LIN {X 0,Y 258.894,Z 466.884,A -85,B 0,C 180,E1 -21997.54,E2 -21997.54} C_VEL
LIN {X 0,Y 258.497,Z 472.697,A -85,B 0,C 180,E1 -21997.806,E2 -21997.806} C_VEL
LIN {X 0,Y 256.025,Z 487.683,A -85,B 0,C 180,E1 -21997.807,E2 -21997.807} C_VEL
LIN {X 0,Y 255.441,Z 492.024,A -85,B 0,C 180,E1 -21997.871,E2 -21997.871} C_VEL
LIN {X 0,Y 249.944,Z 542.974,A -85,B 0,C 180,E1 -21999.352,E2 -21999.352} C_VEL
LIN {X 0,Y 247.16,Z 558.513,A -85,B 0,C 180,E1 -22000.006,E2 -22000.006} C_VEL
LIN {X 0,Y 243.376,Z 573.661,A -85,B 0,C 180,E1 -22000.867,E2 -22000.867} C_VEL
LIN {X 0,Y 238.802,Z 588.296,A -85,B 0,C 180,E1 -22002.002,E2 -22002.002} C_VEL
LIN {X 0,Y 233.418,Z 602.419,A -85,B 0,C 180,E1 -22003.415,E2 -22003.415} C_VEL
LIN {X 0,Y 227.735,Z 615.394,A -85,B 0,C 180,E1 -22005.11,E2 -22005.11} C_VEL
LIN {X 0,Y 221.851,Z 627.382,A -85,B 0,C 180,E1 -22007.08,E2 -22007.08} C_VEL
LIN {X 0,Y 215.808,Z 638.427,A -85,B 0,C 180,E1 -22009.358,E2 -22009.358} C_VEL
LIN {X 0,Y 209.362,Z 649.302,A -85,B 0,C 180,E1 -22012.219,E2 -22012.219} C_VEL
LIN {X 0,Y 202.723,Z 659.642,A -85,B 0,C 180,E1 -22015.711,E2 -22015.711} C_VEL
LIN {X 0,Y 197.738,Z 667.198,A -85,B 0,C 180,E1 -22018.978,E2 -22018.978} C_VEL
LIN {X 0,Y 192.862,Z 674.32,A -85,B 0,C 180,E1 -22022.901,E2 -22022.901} C_VEL
LIN {X 0,Y 188.983,Z 680.037,A -85,B 0,C 180,E1 -22027.015,E2 -22027.015} C_VEL
LIN {X 0,Y 186.775,Z 683.529,A -85,B 0,C 180,E1 -22030.204,E2 -22030.204} C_VEL
LIN {X 0,Y 184.668,Z 687.065,A -85,B 0,C 180,E1 -22034.549,E2 -22034.549} C_VEL
LIN {X 0,Y 183.499,Z 689.425,A -85,B 0,C 180,E1 -22038.959,E2 -22038.959} C_VEL
LIN {X 0,Y 183.209,Z 690.67,A -85,B 0,C 180,E1 -22043.391,E2 -22043.391} C_VEL
LIN {X 0,Y 183.489,Z 690.777,A -85,B 0,C 180,E1 -22047.804,E2 -22047.804} C_VEL
LIN {X 0,Y 183.575,Z 690.376,A -85,B 0,C 180,E1 -22049.999,E2 -22049.999} C_VEL
LIN {X 0,Y 183.501,Z 689.635,A -85,B 0,C 180,E1 -22052.194,E2 -22052.194} C_VEL
LIN {X 0,Y 183.393,Z 688.283,A -85,B 0,C 180,E1 -22054.89,E2 -22054.89} C_VEL
LIN {X 0,Y 183.468,Z 684.438,A -85,B 0,C 180,E1 -22059.925,E2 -22059.925} C_VEL
LIN {X 0,Y 184.277,Z 679.597,A -85,B 0,C 180,E1 -22064.352,E2 -22064.352} C_VEL
LIN {X 0,Y 185.905,Z 673.547,A -85,B 0,C 180,E1 -22068.553,E2 -22068.553} C_VEL
LIN {X 0,Y 188.14,Z 666.3,A -85,B 0,C 180,E1 -22072.512,E2 -22072.512} C_VEL
LIN {X 0,Y 191.186,Z 657.896,A -85,B 0,C 180,E1 -22076.174,E2 -22076.174} C_VEL
LIN {X 0,Y 194.447,Z 648.32,A -85,B 0,C 180,E1 -22079.564,E2 -22079.564} C_VEL
LIN {X 0,Y 198.437,Z 637.302,A -85,B 0,C 180,E1 -22082.69,E2 -22082.69} C_VEL
LIN {X 0,Y 202.681,Z 624.904,A -85,B 0,C 180,E1 -22085.506,E2 -22085.506} C_VEL
LIN {X 0,Y 207.036,Z 611.105,A -85,B 0,C 180,E1 -22087.97,E2 -22087.97} C_VEL
LIN {X 0,Y 210.313,Z 599.494,A -85,B 0,C 180,E1 -22089.627,E2 -22089.627} C_VEL
LIN {X 0,Y 213.614,Z 586.184,A -85,B 0,C 180,E1 -22091.147,E2 -22091.147} C_VEL
LIN {X 0,Y 216.705,Z 571.321,A -85,B 0,C 180,E1 -22092.451,E2 -22092.451} C_VEL
LIN {X 0,Y 219.017,Z 556.883,A -85,B 0,C 180,E1 -22093.384,E2 -22093.384} C_VEL
LIN {X 0,Y 220.649,Z 541.441,A -85,B 0,C 180,E1 -22094.086,E2 -22094.086} C_VEL
LIN {X 0,Y 226.58,Z 457.676,A -85,B 0,C 180,E1 -22096.818,E2 -22096.818} C_VEL
LIN {X 0,Y 221.97,Z 445.741,A -85,B 0,C 180,E1 -22098.326,E2 -22098.326} C_VEL
LIN {X 0,Y 214.721,Z 429.117,A -85,B 0,C 180,E1 -22100.794,E2 -22100.794} C_VEL
LIN {X 0,Y 207.931,Z 415.232,A -85,B 0,C 180,E1 -22103.211,E2 -22103.211} C_VEL
LIN {X 0,Y 200.809,Z 401.844,A -85,B 0,C 180,E1 -22105.947,E2 -22105.947} C_VEL
LIN {X 0,Y 194.594,Z 391.34,A -85,B 0,C 180,E1 -22108.497,E2 -22108.497} C_VEL
LIN {X 0,Y 191.128,Z 385.801,A -85,B 0,C 180,E1 -22110.01,E2 -22110.01} C_VEL
LIN {X 0,Y 189.077,Z 382.495,A -85,B 0,C 180,E1 -22110.953,E2 -22110.953} C_VEL
LIN {X 0,Y 186.429,Z 379.541,A -85,B 0,C 180,E1 -22112.116,E2 -22112.116} C_VEL
LIN {X 0,Y 185.553,Z 376.999,A -85,B 0,C 180,E1 -22112.662,E2 -22112.662} C_VEL
LIN {X 0,Y 185.585,Z 376.991,A -85,B 0,C 180,E1 -22115.383,E2 -22115.383} C_VEL
LIN {X 0,Y 185.672,Z 376.976,A -85,B 0,C 180,E1 -22121.133,E2 -22121.133} C_VEL
LIN {X 0,Y 185.717,Z 376.979,A -85,B 0,C 180,E1 -22124.64,E2 -22124.64} C_VEL
LIN {X 0,Y 185.921,Z 376.902,A -85,B 0,C 180,E1 -22129.36,E2 -22129.36} C_VEL
LIN {X 0,Y 185.958,Z 376.943,A -85,B 0,C 180,E1 -22133.491,E2 -22133.491} C_VEL
LIN {X 0,Y 186.206,Z 376.889,A -85,B 0,C 180,E1 -22137.838,E2 -22137.838} C_VEL
LIN {X 0,Y 186.405,Z 376.87,A -85,B 0,C 180,E1 -22140.001,E2 -22140.001} C_VEL
LIN {X 0,Y 185.925,Z 376.943,A -85,B 0,C 180,E1 -22144.337,E2 -22144.337} C_VEL
LIN {X 0,Y 186.022,Z 376.915,A -85,B 0,C 180,E1 -22148.693,E2 -22148.693} C_VEL
LIN {X 0,Y 185.763,Z 376.965,A -85,B 0,C 180,E1 -22153.121,E2 -22153.121} C_VEL
LIN {X 0,Y 185.673,Z 376.968,A -85,B 0,C 180,E1 -22158.867,E2 -22158.867} C_VEL
LIN {X 0,Y 185.576,Z 376.965,A -85,B 0,C 180,E1 -22164.647,E2 -22164.647} C_VEL
LIN {X 0,Y 185.578,Z 376.992,A -85,B 0,C 180,E1 -22169.494,E2 -22169.494} C_VEL
LIN {X 0,Y 185.499,Z 376.973,A -85,B 0,C 180,E1 -22174.633,E2 -22174.633} C_VEL
LIN {X 0,Y 185.505,Z 376.99,A -85,B 0,C 180,E1 -22177.314,E2 -22177.314} C_VEL
LIN {X 0,Y 185.47,Z 377.001,A -85,B 0,C 180,E1 -22180.726,E2 -22180.726} C_VEL
LIN {X 0,Y 185.459,Z 377.003,A -85,B 0,C 180,E1 -22186.057,E2 -22186.057} C_VEL
LIN {X 0,Y 185.467,Z 376.991,A -85,B 0,C 180,E1 -22189.896,E2 -22189.896} C_VEL
LIN {X 0,Y 185.506,Z 376.986,A -85,B 0,C 180,E1 -22192.713,E2 -22192.713} C_VEL
LIN {X 0,Y 185.534,Z 376.98,A -85,B 0,C 180,E1 -22197.974,E2 -22197.974} C_VEL
LIN {X 0,Y 185.552,Z 376.994,A -85,B 0,C 180,E1 -22200.595,E2 -22200.595} C_VEL
LIN {X 0,Y 185.582,Z 376.98,A -85,B 0,C 180,E1 -22205.383,E2 -22205.383} C_VEL
LIN {X 0,Y 185.594,Z 377.186,A -85,B 0,C 180,E1 -22208.538,E2 -22208.538} C_VEL
LIN {X 0,Y 186.504,Z 379.774,A -85,B 0,C 180,E1 -22209.065,E2 -22209.065} C_VEL
LIN {X 0,Y 188.589,Z 381.975,A -85,B 0,C 180,E1 -22209.979,E2 -22209.979} C_VEL
LIN {X 0,Y 189.237,Z 382.799,A -85,B 0,C 180,E1 -22210.265,E2 -22210.265} C_VEL
LIN {X 0,Y 191.446,Z 386.042,A -85,B 0,C 180,E1 -22211.243,E2 -22211.243} C_VEL
LIN {X 0,Y 192.728,Z 387.647,A -85,B 0,C 180,E1 -22211.774,E2 -22211.774} C_VEL
LIN {X 0,Y 196.707,Z 393.467,A -85,B 0,C 180,E1 -22213.436,E2 -22213.436} C_VEL
LIN {X 0,Y 202.066,Z 401.068,A -85,B 0,C 180,E1 -22215.492,E2 -22215.492} C_VEL
LIN {X 0,Y 208.644,Z 411.142,A -85,B 0,C 180,E1 -22217.858,E2 -22217.858} C_VEL
LIN {X 0,Y 218.699,Z 428.297,A -85,B 0,C 180,E1 -22221.182,E2 -22221.182} C_VEL
LIN {X 0,Y 224.077,Z 439.264,A -85,B 0,C 180,E1 -22222.896,E2 -22222.896} C_VEL
LIN {X 0,Y 226.692,Z 444.585,A -85,B 0,C 180,E1 -22223.685,E2 -22223.685} C_VEL
LIN {X 0,Y 221.003,Z 525.158,A -85,B 0,C 180,E1 -22226.354,E2 -22226.354} C_VEL
LIN {X 0,Y 219.241,Z 540.282,A -85,B 0,C 180,E1 -22227.158,E2 -22227.158} C_VEL
LIN {X 0,Y 216.778,Z 556.065,A -85,B 0,C 180,E1 -22228.375,E2 -22228.375} C_VEL
LIN {X 0,Y 213.955,Z 569.884,A -85,B 0,C 180,E1 -22229.766,E2 -22229.766} C_VEL
LIN {X 0,Y 210.61,Z 583.889,A -85,B 0,C 180,E1 -22231.582,E2 -22231.582} C_VEL
LIN {X 0,Y 207.012,Z 596.7,A -85,B 0,C 180,E1 -22233.651,E2 -22233.651} C_VEL
LIN {X 0,Y 203,Z 609.426,A -85,B 0,C 180,E1 -22236.212,E2 -22236.212} C_VEL
LIN {X 0,Y 199.238,Z 620.577,A -85,B 0,C 180,E1 -22238.995,E2 -22238.995} C_VEL
LIN {X 0,Y 195.131,Z 631.811,A -85,B 0,C 180,E1 -22242.481,E2 -22242.481} C_VEL
LIN {X 0,Y 191.905,Z 640.574,A -85,B 0,C 180,E1 -22245.855,E2 -22245.855} C_VEL
LIN {X 0,Y 189.074,Z 648.331,A -85,B 0,C 180,E1 -22249.545,E2 -22249.545} C_VEL
LIN {X 0,Y 186.876,Z 654.596,A -85,B 0,C 180,E1 -22253.26,E2 -22253.26} C_VEL
LIN {X 0,Y 185.27,Z 659.746,A -85,B 0,C 180,E1 -22257.079,E2 -22257.079} C_VEL
LIN {X 0,Y 184.026,Z 663.921,A -85,B 0,C 180,E1 -22261.037,E2 -22261.037} C_VEL
LIN {X 0,Y 183.21,Z 667.1,A -85,B 0,C 180,E1 -22265.129,E2 -22265.129} C_VEL
LIN {X 0,Y 183.007,Z 669.413,A -85,B 0,C 180,E1 -22269.819,E2 -22269.819} C_VEL
LIN {X 0,Y 183.291,Z 670.312,A -85,B 0,C 180,E1 -22273.646,E2 -22273.646} C_VEL
LIN {X 0,Y 183.797,Z 670.444,A -85,B 0,C 180,E1 -22276.597,E2 -22276.597} C_VEL
LIN {X 0,Y 184.616,Z 670.065,A -85,B 0,C 180,E1 -22279.671,E2 -22279.671} C_VEL
LIN {X 0,Y 185.823,Z 669.085,A -85,B 0,C 180,E1 -22282.76,E2 -22282.76} C_VEL
LIN {X 0,Y 188.251,Z 666.631,A -85,B 0,C 180,E1 -22287.225,E2 -22287.225} C_VEL
LIN {X 0,Y 191.654,Z 662.78,A -85,B 0,C 180,E1 -22291.654,E2 -22291.654} C_VEL
LIN {X 0,Y 195.826,Z 657.743,A -85,B 0,C 180,E1 -22295.762,E2 -22295.762} C_VEL
LIN {X 0,Y 200.527,Z 651.657,A -85,B 0,C 180,E1 -22299.483,E2 -22299.483} C_VEL
LIN {X 0,Y 205.875,Z 644.351,A -85,B 0,C 180,E1 -22302.912,E2 -22302.912} C_VEL
LIN {X 0,Y 211.587,Z 635.885,A -85,B 0,C 180,E1 -22306.055,E2 -22306.055} C_VEL
LIN {X 0,Y 217.343,Z 626.565,A -85,B 0,C 180,E1 -22308.812,E2 -22308.812} C_VEL
LIN {X 0,Y 223.561,Z 615.487,A -85,B 0,C 180,E1 -22311.394,E2 -22311.394} C_VEL
LIN {X 0,Y 229.638,Z 603.29,A -85,B 0,C 180,E1 -22313.63,E2 -22313.63} C_VEL
LIN {X 0,Y 235.175,Z 590.54,A -85,B 0,C 180,E1 -22315.5,E2 -22315.5} C_VEL
LIN {X 0,Y 239.706,Z 578.249,A -85,B 0,C 180,E1 -22316.957,E2 -22316.957} C_VEL
LIN {X 0,Y 244.067,Z 564.231,A -85,B 0,C 180,E1 -22318.246,E2 -22318.246} C_VEL
LIN {X 0,Y 247.639,Z 549.484,A -85,B 0,C 180,E1 -22319.311,E2 -22319.311} C_VEL
LIN {X 0,Y 250.324,Z 534.829,A -85,B 0,C 180,E1 -22320.074,E2 -22320.074} C_VEL
LIN {X 0,Y 252.627,Z 516.015,A -85,B 0,C 180,E1 -22320.717,E2 -22320.717} C_VEL
LIN {X 0,Y 258.11,Z 463.213,A -85,B 0,C 180,E1 -22322.272,E2 -22322.272} C_VEL
LIN {X 0,Y 255.837,Z 458.618,A -85,B 0,C 180,E1 -22323.825,E2 -22323.825} C_VEL
LIN {X 0,Y 252.805,Z 452.119,A -85,B 0,C 180,E1 -22326.308,E2 -22326.308} C_VEL
LIN {X 0,Y 251.193,Z 449.368,A -85,B 0,C 180,E1 -22327.778,E2 -22327.778} C_VEL
LIN {X 0,Y 249.475,Z 446.388,A -85,B 0,C 180,E1 -22329.598,E2 -22329.598} C_VEL
LIN {X 0,Y 247.451,Z 442.793,A -85,B 0,C 180,E1 -22332.401,E2 -22332.401} C_VEL
LIN {X 0,Y 245.547,Z 439.936,A -85,B 0,C 180,E1 -22336.85,E2 -22336.85} C_VEL
LIN {X 0,Y 245.453,Z 439.014,A -85,B 0,C 180,E1 -22337.934,E2 -22337.934} C_VEL
LIN {X 0,Y 245.363,Z 440.064,A -85,B 0,C 180,E1 -22341.586,E2 -22341.586} C_VEL
LIN {X 0,Y 245.757,Z 441.035,A -85,B 0,C 180,E1 -22343.381,E2 -22343.381} C_VEL
LIN {X 0,Y 247.729,Z 446.1,A -85,B 0,C 180,E1 -22347.687,E2 -22347.687} C_VEL
LIN {X 0,Y 250.076,Z 451.667,A -85,B 0,C 180,E1 -22350.753,E2 -22350.753} C_VEL
LIN {X 0,Y 252.319,Z 457.376,A -85,B 0,C 180,E1 -22353.055,E2 -22353.055} C_VEL
LIN {X 0,Y 254.622,Z 463.714,A -85,B 0,C 180,E1 -22355.098,E2 -22355.098} C_VEL
LIN {X 0,Y 257.449,Z 472.109,A -85,B 0,C 180,E1 -22357.257,E2 -22357.257} C_VEL
LIN {X 0,Y 257.008,Z 477.164,A -85,B 0,C 180,E1 -22357.446,E2 -22357.446} C_VEL
LIN {X 0,Y 255.441,Z 492.024,A -85,B 0,C 180,E1 -22357.871,E2 -22357.871} C_VEL
LIN {X 0,Y 254.506,Z 497.876,A -85,B 0,C 180,E1 -22357.886,E2 -22357.886} C_VEL
LIN {X 0,Y 249.984,Z 516.998,A -85,B 0,C 180,E1 -22357.218,E2 -22357.218} C_VEL
LIN {X 0,Y 249.146,Z 522.826,A -85,B 0,C 180,E1 -22357.28,E2 -22357.28} C_VEL
LIN {X 0,Y 246.488,Z 544.542,A -85,B 0,C 180,E1 -22357.949,E2 -22357.949} C_VEL
LIN {X 0,Y 243.261,Z 560.781,A -85,B 0,C 180,E1 -22358.651,E2 -22358.651} C_VEL
LIN {X 0,Y 239.213,Z 575.71,A -85,B 0,C 180,E1 -22359.536,E2 -22359.536} C_VEL
LIN {X 0,Y 234.206,Z 590.658,A -85,B 0,C 180,E1 -22360.737,E2 -22360.737} C_VEL
LIN {X 0,Y 228.684,Z 604.269,A -85,B 0,C 180,E1 -22362.147,E2 -22362.147} C_VEL
LIN {X 0,Y 222.387,Z 617.794,A -85,B 0,C 180,E1 -22363.99,E2 -22363.99} C_VEL
LIN {X 0,Y 215.697,Z 630.347,A -85,B 0,C 180,E1 -22366.18,E2 -22366.18} C_VEL
LIN {X 0,Y 208.568,Z 642.468,A -85,B 0,C 180,E1 -22368.921,E2 -22368.921} C_VEL
LIN {X 0,Y 202.013,Z 652.619,A -85,B 0,C 180,E1 -22371.864,E2 -22371.864} C_VEL
LIN {X 0,Y 196.098,Z 661.158,A -85,B 0,C 180,E1 -22375.009,E2 -22375.009} C_VEL
LIN {X 0,Y 190.324,Z 669.289,A -85,B 0,C 180,E1 -22378.87,E2 -22378.87} C_VEL
LIN {X 0,Y 185.374,Z 675.928,A -85,B 0,C 180,E1 -22382.937,E2 -22382.937} C_VEL
LIN {X 0,Y 181.546,Z 681.214,A -85,B 0,C 180,E1 -22387.224,E2 -22387.224} C_VEL
LIN {X 0,Y 178.786,Z 685.274,A -85,B 0,C 180,E1 -22391.67,E2 -22391.67} C_VEL
LIN {X 0,Y 176.947,Z 688.139,A -85,B 0,C 180,E1 -22396.212,E2 -22396.212} C_VEL
LIN {X 0,Y 176.208,Z 689.84,A -85,B 0,C 180,E1 -22400.819,E2 -22400.819} C_VEL
LIN {X 0,Y 176.26,Z 690.43,A -85,B 0,C 180,E1 -22405.425,E2 -22405.425} C_VEL
LIN {X 0,Y 176.394,Z 690.291,A -85,B 0,C 180,E1 -22407.716,E2 -22407.716} C_VEL
LIN {X 0,Y 176.51,Z 689.846,A -85,B 0,C 180,E1 -22409.999,E2 -22409.999} C_VEL
LIN {X 0,Y 176.411,Z 689.074,A -85,B 0,C 180,E1 -22412.282,E2 -22412.282} C_VEL
LIN {X 0,Y 176.324,Z 687.819,A -85,B 0,C 180,E1 -22414.829,E2 -22414.829} C_VEL
LIN {X 0,Y 176.326,Z 684.745,A -85,B 0,C 180,E1 -22419.173,E2 -22419.173} C_VEL
LIN {X 0,Y 177.002,Z 680.138,A -85,B 0,C 180,E1 -22423.781,E2 -22423.781} C_VEL
LIN {X 0,Y 178.651,Z 674.057,A -85,B 0,C 180,E1 -22428.342,E2 -22428.342} C_VEL
LIN {X 0,Y 181.121,Z 666.318,A -85,B 0,C 180,E1 -22432.831,E2 -22432.831} C_VEL
LIN {X 0,Y 184.232,Z 657.999,A -85,B 0,C 180,E1 -22436.629,E2 -22436.629} C_VEL
LIN {X 0,Y 187.638,Z 648.476,A -85,B 0,C 180,E1 -22440.15,E2 -22440.15} C_VEL
LIN {X 0,Y 191.71,Z 637.625,A -85,B 0,C 180,E1 -22443.358,E2 -22443.358} C_VEL
LIN {X 0,Y 195.682,Z 626.455,A -85,B 0,C 180,E1 -22446.022,E2 -22446.022} C_VEL
LIN {X 0,Y 199.789,Z 614.455,A -85,B 0,C 180,E1 -22448.315,E2 -22448.315} C_VEL
LIN {X 0,Y 203.647,Z 601.464,A -85,B 0,C 180,E1 -22450.32,E2 -22450.32} C_VEL
LIN {X 0,Y 207.234,Z 587.586,A -85,B 0,C 180,E1 -22452.008,E2 -22452.008} C_VEL
LIN {X 0,Y 210.436,Z 572.908,A -85,B 0,C 180,E1 -22453.371,E2 -22453.371} C_VEL
LIN {X 0,Y 213.067,Z 557.48,A -85,B 0,C 180,E1 -22454.418,E2 -22454.418} C_VEL
LIN {X 0,Y 214.774,Z 542.635,A -85,B 0,C 180,E1 -22455.124,E2 -22455.124} C_VEL
LIN {X 0,Y 220.925,Z 459.382,A -85,B 0,C 180,E1 -22457.888,E2 -22457.888} C_VEL
LIN {X 0,Y 212.862,Z 439.507,A -85,B 0,C 180,E1 -22460.691,E2 -22460.691} C_VEL
LIN {X 0,Y 204.972,Z 422.541,A -85,B 0,C 180,E1 -22463.587,E2 -22463.587} C_VEL
LIN {X 0,Y 197.06,Z 407.226,A -85,B 0,C 180,E1 -22466.729,E2 -22466.729} C_VEL
LIN {X 0,Y 190.655,Z 396.248,A -85,B 0,C 180,E1 -22469.479,E2 -22469.479} C_VEL
LIN {X 0,Y 187.522,Z 391.178,A -85,B 0,C 180,E1 -22470.907,E2 -22470.907} C_VEL
LIN {X 0,Y 184.927,Z 387.438,A -85,B 0,C 180,E1 -22472.113,E2 -22472.113} C_VEL
LIN {X 0,Y 182.541,Z 384.257,A -85,B 0,C 180,E1 -22473.258,E2 -22473.258} C_VEL
LIN {X 0,Y 181.864,Z 383.068,A -85,B 0,C 180,E1 -22473.615,E2 -22473.615} C_VEL
LIN {X 0,Y 179.618,Z 380.883,A -85,B 0,C 180,E1 -22474.699,E2 -22474.699} C_VEL
LIN {X 0,Y 178.648,Z 378.396,A -85,B 0,C 180,E1 -22475.289,E2 -22475.289} C_VEL
LIN {X 0,Y 178.542,Z 377.868,A -85,B 0,C 180,E1 -22475.434,E2 -22475.434} C_VEL
LIN {X 0,Y 178.647,Z 377.85,A -85,B 0,C 180,E1 -22481.657,E2 -22481.657} C_VEL
LIN {X 0,Y 178.664,Z 377.83,A -85,B 0,C 180,E1 -22486.349,E2 -22486.349} C_VEL
LIN {X 0,Y 178.935,Z 377.782,A -85,B 0,C 180,E1 -22490.962,E2 -22490.962} C_VEL
LIN {X 0,Y 179.152,Z 377.767,A -85,B 0,C 180,E1 -22497.753,E2 -22497.753} C_VEL
LIN {X 0,Y 179.368,Z 377.745,A -85,B 0,C 180,E1 -22500.001,E2 -22500.001} C_VEL
LIN {X 0,Y 178.873,Z 377.819,A -85,B 0,C 180,E1 -22504.508,E2 -22504.508} C_VEL
LIN {X 0,Y 178.973,Z 377.796,A -85,B 0,C 180,E1 -22509.038,E2 -22509.038} C_VEL
LIN {X 0,Y 178.68,Z 377.842,A -85,B 0,C 180,E1 -22513.651,E2 -22513.651} C_VEL
LIN {X 0,Y 178.621,Z 377.849,A -85,B 0,C 180,E1 -22519.216,E2 -22519.216} C_VEL
LIN {X 0,Y 178.519,Z 377.839,A -85,B 0,C 180,E1 -22525.115,E2 -22525.115} C_VEL
LIN {X 0,Y 178.5,Z 377.875,A -85,B 0,C 180,E1 -22530.788,E2 -22530.788} C_VEL
LIN {X 0,Y 178.484,Z 377.847,A -85,B 0,C 180,E1 -22534.221,E2 -22534.221} C_VEL
LIN {X 0,Y 178.395,Z 377.889,A -85,B 0,C 180,E1 -22539.076,E2 -22539.076} C_VEL
LIN {X 0,Y 178.397,Z 377.866,A -85,B 0,C 180,E1 -22542.047,E2 -22542.047} C_VEL
LIN {X 0,Y 178.393,Z 377.869,A -85,B 0,C 180,E1 -22545.166,E2 -22545.166} C_VEL
LIN {X 0,Y 178.403,Z 377.885,A -85,B 0,C 180,E1 -22548.461,E2 -22548.461} C_VEL
LIN {X 0,Y 178.423,Z 377.881,A -85,B 0,C 180,E1 -22553.784,E2 -22553.784} C_VEL
LIN {X 0,Y 178.485,Z 377.868,A -85,B 0,C 180,E1 -22556.548,E2 -22556.548} C_VEL
LIN {X 0,Y 178.451,Z 377.882,A -85,B 0,C 180,E1 -22561.798,E2 -22561.798} C_VEL
LIN {X 0,Y 178.52,Z 377.862,A -85,B 0,C 180,E1 -22565.737,E2 -22565.737} C_VEL
LIN {X 0,Y 179.413,Z 380.567,A -85,B 0,C 180,E1 -22566.337,E2 -22566.337} C_VEL
LIN {X 0,Y 181.466,Z 382.798,A -85,B 0,C 180,E1 -22567.332,E2 -22567.332} C_VEL
LIN {X 0,Y 182.218,Z 383.521,A -85,B 0,C 180,E1 -22567.687,E2 -22567.687} C_VEL
LIN {X 0,Y 184.171,Z 386.748,A -85,B 0,C 180,E1 -22568.686,E2 -22568.686} C_VEL
LIN {X 0,Y 185.81,Z 388.531,A -85,B 0,C 180,E1 -22569.427,E2 -22569.427} C_VEL
LIN {X 0,Y 188.431,Z 392.16,A -85,B 0,C 180,E1 -22570.616,E2 -22570.616} C_VEL
LIN {X 0,Y 197.691,Z 405.469,A -85,B 0,C 180,E1 -22574.477,E2 -22574.477} C_VEL
LIN {X 0,Y 204.48,Z 416.004,A -85,B 0,C 180,E1 -22577.014,E2 -22577.014} C_VEL
LIN {X 0,Y 214.143,Z 432.761,A -85,B 0,C 180,E1 -22580.364,E2 -22580.364} C_VEL
LIN {X 0,Y 221.046,Z 446.985,A -85,B 0,C 180,E1 -22582.624,E2 -22582.624} C_VEL
LIN {X 0,Y 215.267,Z 525.461,A -85,B 0,C 180,E1 -22585.261,E2 -22585.261} C_VEL
LIN {X 0,Y 213.393,Z 541.006,A -85,B 0,C 180,E1 -22586.106,E2 -22586.106} C_VEL
LIN {X 0,Y 211.091,Z 555.393,A -85,B 0,C 180,E1 -22587.222,E2 -22587.222} C_VEL
LIN {X 0,Y 207.872,Z 570.702,A -85,B 0,C 180,E1 -22588.79,E2 -22588.79} C_VEL
LIN {X 0,Y 204.407,Z 584.636,A -85,B 0,C 180,E1 -22590.645,E2 -22590.645} C_VEL
LIN {X 0,Y 200.676,Z 597.405,A -85,B 0,C 180,E1 -22592.761,E2 -22592.761} C_VEL
LIN {X 0,Y 196.539,Z 610.109,A -85,B 0,C 180,E1 -22595.398,E2 -22595.398} C_VEL
LIN {X 0,Y 192.43,Z 621.712,A -85,B 0,C 180,E1 -22598.401,E2 -22598.401} C_VEL
LIN {X 0,Y 188.409,Z 632.382,A -85,B 0,C 180,E1 -22601.84,E2 -22601.84} C_VEL
LIN {X 0,Y 184.955,Z 641.345,A -85,B 0,C 180,E1 -22605.427,E2 -22605.427} C_VEL
LIN {X 0,Y 182.123,Z 648.872,A -85,B 0,C 180,E1 -22609.149,E2 -22609.149} C_VEL
LIN {X 0,Y 179.824,Z 655.13,A -85,B 0,C 180,E1 -22613.007,E2 -22613.007} C_VEL
LIN {X 0,Y 178.17,Z 660.26,A -85,B 0,C 180,E1 -22616.977,E2 -22616.977} C_VEL
LIN {X 0,Y 176.891,Z 664.415,A -85,B 0,C 180,E1 -22621.099,E2 -22621.099} C_VEL
LIN {X 0,Y 176.297,Z 666.609,A -85,B 0,C 180,E1 -22623.926,E2 -22623.926} C_VEL
LIN {X 0,Y 175.946,Z 668.452,A -85,B 0,C 180,E1 -22626.975,E2 -22626.975} C_VEL
LIN {X 0,Y 175.961,Z 670.003,A -85,B 0,C 180,E1 -22630.634,E2 -22630.634} C_VEL
LIN {X 0,Y 176.538,Z 670.91,A -85,B 0,C 180,E1 -22635.774,E2 -22635.774} C_VEL
LIN {X 0,Y 177.874,Z 670.433,A -85,B 0,C 180,E1 -22640.788,E2 -22640.788} C_VEL
LIN {X 0,Y 179.838,Z 668.849,A -85,B 0,C 180,E1 -22645.154,E2 -22645.154} C_VEL
LIN {X 0,Y 183.09,Z 665.712,A -85,B 0,C 180,E1 -22650.064,E2 -22650.064} C_VEL
LIN {X 0,Y 186.985,Z 661.483,A -85,B 0,C 180,E1 -22654.433,E2 -22654.433} C_VEL
LIN {X 0,Y 191.705,Z 656.042,A -85,B 0,C 180,E1 -22658.493,E2 -22658.493} C_VEL
LIN {X 0,Y 196.988,Z 649.526,A -85,B 0,C 180,E1 -22662.185,E2 -22662.185} C_VEL
LIN {X 0,Y 203.111,Z 641.488,A -85,B 0,C 180,E1 -22665.665,E2 -22665.665} C_VEL
LIN {X 0,Y 209.522,Z 632.045,A -85,B 0,C 180,E1 -22668.879,E2 -22668.879} C_VEL
LIN {X 0,Y 216.08,Z 621.491,A -85,B 0,C 180,E1 -22671.66,E2 -22671.66} C_VEL
LIN {X 0,Y 222.382,Z 610.196,A -85,B 0,C 180,E1 -22674.004,E2 -22674.004} C_VEL
LIN {X 0,Y 228.469,Z 597.665,A -85,B 0,C 180,E1 -22676.072,E2 -22676.072} C_VEL
LIN {X 0,Y 233.908,Z 584.523,A -85,B 0,C 180,E1 -22677.801,E2 -22677.801} C_VEL
LIN {X 0,Y 238.975,Z 570.102,A -85,B 0,C 180,E1 -22679.254,E2 -22679.254} C_VEL
LIN {X 0,Y 242.928,Z 555.944,A -85,B 0,C 180,E1 -22680.39,E2 -22680.39} C_VEL
LIN {X 0,Y 246.221,Z 540.757,A -85,B 0,C 180,E1 -22681.281,E2 -22681.281} C_VEL
LIN {X 0,Y 248.541,Z 525.48,A -85,B 0,C 180,E1 -22681.899,E2 -22681.899} C_VEL
LIN {X 0,Y 254.873,Z 467.067,A -85,B 0,C 180,E1 -22683.605,E2 -22683.605} C_VEL
LIN {X 0,Y 250.885,Z 458.365,A -85,B 0,C 180,E1 -22686.935,E2 -22686.935} C_VEL
LIN {X 0,Y 249.267,Z 455.437,A -85,B 0,C 180,E1 -22688.559,E2 -22688.559} C_VEL
LIN {X 0,Y 247.792,Z 452.807,A -85,B 0,C 180,E1 -22690.245,E2 -22690.245} C_VEL
LIN {X 0,Y 246.195,Z 449.703,A -85,B 0,C 180,E1 -22692.642,E2 -22692.642} C_VEL
LIN {X 0,Y 244.456,Z 446.991,A -85,B 0,C 180,E1 -22696.927,E2 -22696.927} C_VEL
LIN {X 0,Y 244.33,Z 446.02,A -85,B 0,C 180,E1 -22698.335,E2 -22698.335} C_VEL
LIN {X 0,Y 244.55,Z 447.734,A -85,B 0,C 180,E1 -22702.911,E2 -22702.911} C_VEL
LIN {X 0,Y 246.445,Z 453.026,A -85,B 0,C 180,E1 -22707.434,E2 -22707.434} C_VEL
LIN {X 0,Y 248.374,Z 458.128,A -85,B 0,C 180,E1 -22710.173,E2 -22710.173} C_VEL
LIN {X 0,Y 250.507,Z 463.957,A -85,B 0,C 180,E1 -22712.547,E2 -22712.547} C_VEL
LIN {X 0,Y 252.807,Z 470.915,A -85,B 0,C 180,E1 -22714.711,E2 -22714.711} C_VEL
LIN {X 0,Y 254.29,Z 475.637,A -85,B 0,C 180,E1 -22715.956,E2 -22715.956} C_VEL
LIN {X 0,Y 249.146,Z 522.826,A -85,B 0,C 180,E1 -22717.28,E2 -22717.28} C_VEL
LIN {X 0,Y 248.312,Z 528.647,A -85,B 0,C 180,E1 -22717.339,E2 -22717.339} C_VEL
LIN {X 0,Y 243.806,Z 545.746,A -85,B 0,C 180,E1 -22716.754,E2 -22716.754} C_VEL
LIN {X 0,Y 242.284,Z 551.476,A -85,B 0,C 180,E1 -22716.741,E2 -22716.741} C_VEL
LIN {X 0,Y 241.857,Z 553.389,A -85,B 0,C 180,E1 -22716.809,E2 -22716.809} C_VEL
LIN {X 0,Y 238.195,Z 568.177,A -85,B 0,C 180,E1 -22717.537,E2 -22717.537} C_VEL
LIN {X 0,Y 234.245,Z 580.933,A -85,B 0,C 180,E1 -22718.387,E2 -22718.387} C_VEL
LIN {X 0,Y 229.118,Z 594.693,A -85,B 0,C 180,E1 -22719.583,E2 -22719.583} C_VEL
LIN {X 0,Y 223.486,Z 607.466,A -85,B 0,C 180,E1 -22720.997,E2 -22720.997} C_VEL
LIN {X 0,Y 217.057,Z 620.299,A -85,B 0,C 180,E1 -22722.839,E2 -22722.839} C_VEL
LIN {X 0,Y 210.696,Z 631.511,A -85,B 0,C 180,E1 -22724.86,E2 -22724.86} C_VEL
LIN {X 0,Y 203.309,Z 643.323,A -85,B 0,C 180,E1 -22727.616,E2 -22727.616} C_VEL
LIN {X 0,Y 196.49,Z 653.209,A -85,B 0,C 180,E1 -22730.588,E2 -22730.588} C_VEL
LIN {X 0,Y 189.512,Z 662.689,A -85,B 0,C 180,E1 -22734.261,E2 -22734.261} C_VEL
LIN {X 0,Y 184.24,Z 669.539,A -85,B 0,C 180,E1 -22737.72,E2 -22737.72} C_VEL
LIN {X 0,Y 179.028,Z 675.999,A -85,B 0,C 180,E1 -22741.895,E2 -22741.895} C_VEL
LIN {X 0,Y 174.962,Z 681.16,A -85,B 0,C 180,E1 -22746.315,E2 -22746.315} C_VEL
LIN {X 0,Y 171.978,Z 685.098,A -85,B 0,C 180,E1 -22750.917,E2 -22750.917} C_VEL
LIN {X 0,Y 169.998,Z 687.881,A -85,B 0,C 180,E1 -22755.637,E2 -22755.637} C_VEL
LIN {X 0,Y 169.135,Z 689.495,A -85,B 0,C 180,E1 -22760.431,E2 -22760.431} C_VEL
LIN {X 0,Y 169.174,Z 689.981,A -85,B 0,C 180,E1 -22765.575,E2 -22765.575} C_VEL
LIN {X 0,Y 169.445,Z 689.308,A -85,B 0,C 180,E1 -22769.999,E2 -22769.999} C_VEL
LIN {X 0,Y 169.254,Z 687.346,A -85,B 0,C 180,E1 -22774.763,E2 -22774.763} C_VEL
LIN {X 0,Y 169.276,Z 684.052,A -85,B 0,C 180,E1 -22779.558,E2 -22779.558} C_VEL
LIN {X 0,Y 170.038,Z 679.349,A -85,B 0,C 180,E1 -22784.358,E2 -22784.358} C_VEL
LIN {X 0,Y 171.824,Z 673.155,A -85,B 0,C 180,E1 -22789.099,E2 -22789.099} C_VEL
LIN {X 0,Y 174.49,Z 665.277,A -85,B 0,C 180,E1 -22793.751,E2 -22793.751} C_VEL
LIN {X 0,Y 177.825,Z 656.836,A -85,B 0,C 180,E1 -22797.669,E2 -22797.669} C_VEL
LIN {X 0,Y 181.755,Z 646.312,A -85,B 0,C 180,E1 -22801.575,E2 -22801.575} C_VEL
LIN {X 0,Y 185.72,Z 636.122,A -85,B 0,C 180,E1 -22804.584,E2 -22804.584} C_VEL
LIN {X 0,Y 190.317,Z 623.63,A -85,B 0,C 180,E1 -22807.538,E2 -22807.538} C_VEL
LIN {X 0,Y 194.541,Z 611.124,A -85,B 0,C 180,E1 -22809.883,E2 -22809.883} C_VEL
LIN {X 0,Y 198.164,Z 599.118,A -85,B 0,C 180,E1 -22811.679,E2 -22811.679} C_VEL
LIN {X 0,Y 201.976,Z 584.54,A -85,B 0,C 180,E1 -22813.409,E2 -22813.409} C_VEL
LIN {X 0,Y 205.31,Z 569.469,A -85,B 0,C 180,E1 -22814.738,E2 -22814.738} C_VEL
LIN {X 0,Y 207.608,Z 555.502,A -85,B 0,C 180,E1 -22815.652,E2 -22815.652} C_VEL
LIN {X 0,Y 209.211,Z 541.118,A -85,B 0,C 180,E1 -22816.326,E2 -22816.326} C_VEL
LIN {X 0,Y 215.317,Z 461.987,A -85,B 0,C 180,E1 -22818.982,E2 -22818.982} C_VEL
LIN {X 0,Y 214.514,Z 459.403,A -85,B 0,C 180,E1 -22819.295,E2 -22819.295} C_VEL
LIN {X 0,Y 207.41,Z 441.938,A -85,B 0,C 180,E1 -22821.879,E2 -22821.879} C_VEL
LIN {X 0,Y 199.863,Z 425.501,A -85,B 0,C 180,E1 -22824.822,E2 -22824.822} C_VEL
LIN {X 0,Y 192.168,Z 410.605,A -85,B 0,C 180,E1 -22828.043,E2 -22828.043} C_VEL
LIN {X 0,Y 185.106,Z 398.223,A -85,B 0,C 180,E1 -22831.282,E2 -22831.282} C_VEL
LIN {X 0,Y 181.421,Z 392.942,A -85,B 0,C 180,E1 -22833.055,E2 -22833.055} C_VEL
LIN {X 0,Y 178.917,Z 389.315,A -85,B 0,C 180,E1 -22834.342,E2 -22834.342} C_VEL
LIN {X 0,Y 176.159,Z 386.19,A -85,B 0,C 180,E1 -22835.731,E2 -22835.731} C_VEL
LIN {X 0,Y 174.891,Z 383.951,A -85,B 0,C 180,E1 -22836.464,E2 -22836.464} C_VEL
LIN {X 0,Y 172.666,Z 381.903,A -85,B 0,C 180,E1 -22837.648,E2 -22837.648} C_VEL
LIN {X 0,Y 171.584,Z 379.493,A -85,B 0,C 180,E1 -22838.369,E2 -22838.369} C_VEL
LIN {X 0,Y 171.467,Z 378.746,A -85,B 0,C 180,E1 -22838.576,E2 -22838.576} C_VEL
LIN {X 0,Y 171.576,Z 378.733,A -85,B 0,C 180,E1 -22840.872,E2 -22840.872} C_VEL
LIN {X 0,Y 171.591,Z 378.719,A -85,B 0,C 180,E1 -22845.775,E2 -22845.775} C_VEL
LIN {X 0,Y 171.87,Z 378.656,A -85,B 0,C 180,E1 -22850.587,E2 -22850.587} C_VEL
LIN {X 0,Y 171.82,Z 378.705,A -85,B 0,C 180,E1 -22855.308,E2 -22855.308} C_VEL
LIN {X 0,Y 172.331,Z 378.62,A -85,B 0,C 180,E1 -22860.001,E2 -22860.001} C_VEL
LIN {X 0,Y 171.823,Z 378.694,A -85,B 0,C 180,E1 -22864.693,E2 -22864.693} C_VEL
LIN {X 0,Y 171.906,Z 378.679,A -85,B 0,C 180,E1 -22869.413,E2 -22869.413} C_VEL
LIN {X 0,Y 171.592,Z 378.716,A -85,B 0,C 180,E1 -22874.227,E2 -22874.227} C_VEL
LIN {X 0,Y 171.54,Z 378.734,A -85,B 0,C 180,E1 -22879.561,E2 -22879.561} C_VEL
LIN {X 0,Y 171.458,Z 378.716,A -85,B 0,C 180,E1 -22885.61,E2 -22885.61} C_VEL
LIN {X 0,Y 171.458,Z 378.754,A -85,B 0,C 180,E1 -22890.598,E2 -22890.598} C_VEL
LIN {X 0,Y 171.392,Z 378.728,A -85,B 0,C 180,E1 -22895.036,E2 -22895.036} C_VEL
LIN {X 0,Y 171.357,Z 378.764,A -85,B 0,C 180,E1 -22898.809,E2 -22898.809} C_VEL
LIN {X 0,Y 171.32,Z 378.741,A -85,B 0,C 180,E1 -22904.219,E2 -22904.219} C_VEL
LIN {X 0,Y 171.335,Z 378.76,A -85,B 0,C 180,E1 -22908.983,E2 -22908.983} C_VEL
LIN {X 0,Y 171.365,Z 378.741,A -85,B 0,C 180,E1 -22912.037,E2 -22912.037} C_VEL
LIN {X 0,Y 171.399,Z 378.762,A -85,B 0,C 180,E1 -22915.094,E2 -22915.094} C_VEL
LIN {X 0,Y 171.414,Z 378.754,A -85,B 0,C 180,E1 -22920.529,E2 -22920.529} C_VEL
LIN {X 0,Y 171.383,Z 378.754,A -85,B 0,C 180,E1 -22922.569,E2 -22922.569} C_VEL
LIN {X 0,Y 172.291,Z 381.408,A -85,B 0,C 180,E1 -22923.248,E2 -22923.248} C_VEL
LIN {X 0,Y 174.3,Z 383.589,A -85,B 0,C 180,E1 -22924.366,E2 -22924.366} C_VEL
LIN {X 0,Y 175.288,Z 384.409,A -85,B 0,C 180,E1 -22924.875,E2 -22924.875} C_VEL
LIN {X 0,Y 177.084,Z 387.484,A -85,B 0,C 180,E1 -22925.899,E2 -22925.899} C_VEL
LIN {X 0,Y 179.077,Z 389.677,A -85,B 0,C 180,E1 -22926.894,E2 -22926.894} C_VEL
LIN {X 0,Y 181.671,Z 393.292,A -85,B 0,C 180,E1 -22928.197,E2 -22928.197} C_VEL
LIN {X 0,Y 186.339,Z 399.799,A -85,B 0,C 180,E1 -22930.404,E2 -22930.404} C_VEL
LIN {X 0,Y 193.888,Z 410.727,A -85,B 0,C 180,E1 -22933.632,E2 -22933.632} C_VEL
LIN {X 0,Y 200.482,Z 421.216,A -85,B 0,C 180,E1 -22936.222,E2 -22936.222} C_VEL
LIN {X 0,Y 209.6,Z 437.241,A -85,B 0,C 180,E1 -22939.51,E2 -22939.51} C_VEL
LIN {X 0,Y 214.353,Z 447.151,A -85,B 0,C 180,E1 -22941.146,E2 -22941.146} C_VEL
LIN {X 0,Y 215.433,Z 449.385,A -85,B 0,C 180,E1 -22941.502,E2 -22941.502} C_VEL
LIN {X 0,Y 209.565,Z 526.05,A -85,B 0,C 180,E1 -22944.127,E2 -22944.127} C_VEL
LIN {X 0,Y 207.671,Z 541.225,A -85,B 0,C 180,E1 -22944.965,E2 -22944.965} C_VEL
LIN {X 0,Y 205.146,Z 556.418,A -85,B 0,C 180,E1 -22946.174,E2 -22946.174} C_VEL
LIN {X 0,Y 201.796,Z 571.693,A -85,B 0,C 180,E1 -22947.788,E2 -22947.788} C_VEL
LIN {X 0,Y 198.071,Z 585.946,A -85,B 0,C 180,E1 -22949.747,E2 -22949.747} C_VEL
LIN {X 0,Y 193.938,Z 599.39,A -85,B 0,C 180,E1 -22952.078,E2 -22952.078} C_VEL
LIN {X 0,Y 189.797,Z 611.558,A -85,B 0,C 180,E1 -22954.726,E2 -22954.726} C_VEL
LIN {X 0,Y 185.853,Z 622.282,A -85,B 0,C 180,E1 -22957.606,E2 -22957.606} C_VEL
LIN {X 0,Y 181.678,Z 632.928,A -85,B 0,C 180,E1 -22961.153,E2 -22961.153} C_VEL
LIN {X 0,Y 178.114,Z 641.86,A -85,B 0,C 180,E1 -22964.862,E2 -22964.862} C_VEL
LIN {X 0,Y 175.172,Z 649.374,A -85,B 0,C 180,E1 -22968.722,E2 -22968.722} C_VEL
LIN {X 0,Y 172.784,Z 655.621,A -85,B 0,C 180,E1 -22972.733,E2 -22972.733} C_VEL
LIN {X 0,Y 171.071,Z 660.736,A -85,B 0,C 180,E1 -22976.867,E2 -22976.867} C_VEL
LIN {X 0,Y 169.755,Z 664.881,A -85,B 0,C 180,E1 -22981.165,E2 -22981.165} C_VEL
LIN {X 0,Y 168.941,Z 668.049,A -85,B 0,C 180,E1 -22985.621,E2 -22985.621} C_VEL
LIN {X 0,Y 168.813,Z 669.549,A -85,B 0,C 180,E1 -22988.645,E2 -22988.645} C_VEL
LIN {X 0,Y 168.939,Z 670.6,A -85,B 0,C 180,E1 -22991.731,E2 -22991.731} C_VEL
LIN {X 0,Y 169.333,Z 671.225,A -85,B 0,C 180,E1 -22995.123,E2 -22995.123} C_VEL
LIN {X 0,Y 170.073,Z 671.307,A -85,B 0,C 180,E1 -22998.609,E2 -22998.609} C_VEL
LIN {X 0,Y 171.202,Z 670.772,A -85,B 0,C 180,E1 -23001.991,E2 -23001.991} C_VEL
LIN {X 0,Y 172.732,Z 669.679,A -85,B 0,C 180,E1 -23005.275,E2 -23005.275} C_VEL
LIN {X 0,Y 174.659,Z 668.074,A -85,B 0,C 180,E1 -23008.459,E2 -23008.459} C_VEL
LIN {X 0,Y 178.307,Z 664.66,A -85,B 0,C 180,E1 -23013.015,E2 -23013.015} C_VEL
LIN {X 0,Y 182.9,Z 659.953,A -85,B 0,C 180,E1 -23017.402,E2 -23017.402} C_VEL
LIN {X 0,Y 188.429,Z 653.83,A -85,B 0,C 180,E1 -23021.578,E2 -23021.578} C_VEL
LIN {X 0,Y 194.691,Z 646.371,A -85,B 0,C 180,E1 -23025.363,E2 -23025.363} C_VEL
LIN {X 0,Y 201.29,Z 637.705,A -85,B 0,C 180,E1 -23028.749,E2 -23028.749} C_VEL
LIN {X 0,Y 207.838,Z 628.229,A -85,B 0,C 180,E1 -23031.657,E2 -23031.657} C_VEL
LIN {X 0,Y 214.288,Z 617.93,A -85,B 0,C 180,E1 -23034.126,E2 -23034.126} C_VEL
LIN {X 0,Y 220.782,Z 606.189,A -85,B 0,C 180,E1 -23036.349,E2 -23036.349} C_VEL
LIN {X 0,Y 226.794,Z 593.77,A -85,B 0,C 180,E1 -23038.224,E2 -23038.224} C_VEL
LIN {X 0,Y 231.929,Z 581.34,A -85,B 0,C 180,E1 -23039.739,E2 -23039.739} C_VEL
LIN {X 0,Y 236.792,Z 567.288,A -85,B 0,C 180,E1 -23041.062,E2 -23041.062} C_VEL
LIN {X 0,Y 240.565,Z 553.534,A -85,B 0,C 180,E1 -23042.092,E2 -23042.092} C_VEL
LIN {X 0,Y 243.818,Z 537.95,A -85,B 0,C 180,E1 -23042.943,E2 -23042.943} C_VEL
LIN {X 0,Y 246.177,Z 521.343,A -85,B 0,C 180,E1 -23043.53,E2 -23043.53} C_VEL
LIN {X 0,Y 251.822,Z 471.264,A -85,B 0,C 180,E1 -23044.987,E2 -23044.987} C_VEL
LIN {X 0,Y 248.952,Z 464.458,A -85,B 0,C 180,E1 -23047.672,E2 -23047.672} C_VEL
LIN {X 0,Y 246.425,Z 459.648,A -85,B 0,C 180,E1 -23050.565,E2 -23050.565} C_VEL
LIN {X 0,Y 244.873,Z 456.592,A -85,B 0,C 180,E1 -23052.986,E2 -23052.986} C_VEL
LIN {X 0,Y 243.299,Z 453.616,A -85,B 0,C 180,E1 -23057.587,E2 -23057.587} C_VEL
LIN {X 0,Y 243.228,Z 453.076,A -85,B 0,C 180,E1 -23058.532,E2 -23058.532} C_VEL
LIN {X 0,Y 243.412,Z 454.748,A -85,B 0,C 180,E1 -23062.739,E2 -23062.739} C_VEL
LIN {X 0,Y 245.076,Z 459.783,A -85,B 0,C 180,E1 -23067.036,E2 -23067.036} C_VEL
LIN {X 0,Y 246.655,Z 464.449,A -85,B 0,C 180,E1 -23069.531,E2 -23069.531} C_VEL
LIN {X 0,Y 248.654,Z 470.357,A -85,B 0,C 180,E1 -23071.952,E2 -23071.952} C_VEL
LIN {X 0,Y 251.034,Z 478.202,A -85,B 0,C 180,E1 -23074.346,E2 -23074.346} C_VEL
LIN {X 0,Y 251.229,Z 478.949,A -85,B 0,C 180,E1 -23074.538,E2 -23074.538} C_VEL
LIN {X 0,Y 243.979,Z 541.533,A -85,B 0,C 180,E1 -23076.325,E2 -23076.325} C_VEL
LIN {X 0,Y 241.857,Z 553.389,A -85,B 0,C 180,E1 -23076.809,E2 -23076.809} C_VEL
LIN {X 0,Y 240.276,Z 559.09,A -85,B 0,C 180,E1 -23076.903,E2 -23076.903} C_VEL
LIN {X 0,Y 236.593,Z 568.281,A -85,B 0,C 180,E1 -23076.746,E2 -23076.746} C_VEL
LIN {X 0,Y 232.591,Z 577.366,A -85,B 0,C 180,E1 -23076.691,E2 -23076.691} C_VEL
LIN {X 0,Y 230.472,Z 582.682,A -85,B 0,C 180,E1 -23076.952,E2 -23076.952} C_VEL
LIN {X 0,Y 224.745,Z 597.03,A -85,B 0,C 180,E1 -23078.215,E2 -23078.215} C_VEL
LIN {X 0,Y 218.371,Z 610.556,A -85,B 0,C 180,E1 -23079.79,E2 -23079.79} C_VEL
LIN {X 0,Y 211.362,Z 623.479,A -85,B 0,C 180,E1 -23081.754,E2 -23081.754} C_VEL
LIN {X 0,Y 204.682,Z 634.344,A -85,B 0,C 180,E1 -23083.857,E2 -23083.857} C_VEL
LIN {X 0,Y 198.162,Z 644.124,A -85,B 0,C 180,E1 -23086.243,E2 -23086.243} C_VEL
LIN {X 0,Y 191.086,Z 653.824,A -85,B 0,C 180,E1 -23089.243,E2 -23089.243} C_VEL
LIN {X 0,Y 183.777,Z 663.046,A -85,B 0,C 180,E1 -23092.963,E2 -23092.963} C_VEL
LIN {X 0,Y 178.231,Z 669.805,A -85,B 0,C 180,E1 -23096.491,E2 -23096.491} C_VEL
LIN {X 0,Y 172.748,Z 676.122,A -85,B 0,C 180,E1 -23100.776,E2 -23100.776} C_VEL
LIN {X 0,Y 168.415,Z 681.118,A -85,B 0,C 180,E1 -23105.335,E2 -23105.335} C_VEL
LIN {X 0,Y 165.206,Z 684.928,A -85,B 0,C 180,E1 -23110.102,E2 -23110.102} C_VEL
LIN {X 0,Y 163.071,Z 687.6,A -85,B 0,C 180,E1 -23115.013,E2 -23115.013} C_VEL
LIN {X 0,Y 162.086,Z 689.153,A -85,B 0,C 180,E1 -23120.011,E2 -23120.011} C_VEL
LIN {X 0,Y 162.097,Z 689.535,A -85,B 0,C 180,E1 -23125.706,E2 -23125.706} C_VEL
LIN {X 0,Y 162.381,Z 688.765,A -85,B 0,C 180,E1 -23129.999,E2 -23129.999} C_VEL
LIN {X 0,Y 162.164,Z 686.693,A -85,B 0,C 180,E1 -23134.971,E2 -23134.971} C_VEL
LIN {X 0,Y 162.243,Z 683.29,A -85,B 0,C 180,E1 -23139.977,E2 -23139.977} C_VEL
LIN {X 0,Y 163.103,Z 678.482,A -85,B 0,C 180,E1 -23144.982,E2 -23144.982} C_VEL
LIN {X 0,Y 165.034,Z 672.158,A -85,B 0,C 180,E1 -23149.917,E2 -23149.917} C_VEL
LIN {X 0,Y 167.924,Z 664.117,A -85,B 0,C 180,E1 -23154.74,E2 -23154.74} C_VEL
LIN {X 0,Y 171.445,Z 655.529,A -85,B 0,C 180,E1 -23158.793,E2 -23158.793} C_VEL
LIN {X 0,Y 175.278,Z 645.738,A -85,B 0,C 180,E1 -23162.504,E2 -23162.504} C_VEL
LIN {X 0,Y 179.824,Z 634.43,A -85,B 0,C 180,E1 -23165.889,E2 -23165.889} C_VEL
LIN {X 0,Y 184.235,Z 622.847,A -85,B 0,C 180,E1 -23168.656,E2 -23168.656} C_VEL
LIN {X 0,Y 188.605,Z 610.27,A -85,B 0,C 180,E1 -23171.052,E2 -23171.052} C_VEL
LIN {X 0,Y 192.122,Z 598.974,A -85,B 0,C 180,E1 -23172.773,E2 -23172.773} C_VEL
LIN {X 0,Y 195.823,Z 585.502,A -85,B 0,C 180,E1 -23174.413,E2 -23174.413} C_VEL
LIN {X 0,Y 199.211,Z 570.823,A -85,B 0,C 180,E1 -23175.774,E2 -23175.774} C_VEL
LIN {X 0,Y 201.687,Z 556.639,A -85,B 0,C 180,E1 -23176.759,E2 -23176.759} C_VEL
LIN {X 0,Y 203.502,Z 541.82,A -85,B 0,C 180,E1 -23177.485,E2 -23177.485} C_VEL
LIN {X 0,Y 209.732,Z 463.575,A -85,B 0,C 180,E1 -23180.171,E2 -23180.171} C_VEL
LIN {X 0,Y 202.849,Z 446.181,A -85,B 0,C 180,E1 -23182.818,E2 -23182.818} C_VEL
LIN {X 0,Y 195.507,Z 429.996,A -85,B 0,C 180,E1 -23185.798,E2 -23185.798} C_VEL
LIN {X 0,Y 188.497,Z 416.071,A -85,B 0,C 180,E1 -23188.897,E2 -23188.897} C_VEL
LIN {X 0,Y 181.496,Z 403.535,A -85,B 0,C 180,E1 -23192.246,E2 -23192.246} C_VEL
LIN {X 0,Y 177.871,Z 398.295,A -85,B 0,C 180,E1 -23194.082,E2 -23194.082} C_VEL
LIN {X 0,Y 174.943,Z 394.349,A -85,B 0,C 180,E1 -23195.605,E2 -23195.605} C_VEL
LIN {X 0,Y 172.353,Z 390.752,A -85,B 0,C 180,E1 -23197.051,E2 -23197.051} C_VEL
LIN {X 0,Y 171.107,Z 389.357,A -85,B 0,C 180,E1 -23197.751,E2 -23197.751} C_VEL
LIN {X 0,Y 168.951,Z 386.513,A -85,B 0,C 180,E1 -23199.055,E2 -23199.055} C_VEL
LIN {X 0,Y 168.05,Z 384.945,A -85,B 0,C 180,E1 -23199.658,E2 -23199.658} C_VEL
LIN {X 0,Y 165.73,Z 382.779,A -85,B 0,C 180,E1 -23201.096,E2 -23201.096} C_VEL
LIN {X 0,Y 164.666,Z 380.486,A -85,B 0,C 180,E1 -23201.895,E2 -23201.895} C_VEL
LIN {X 0,Y 164.497,Z 379.612,A -85,B 0,C 180,E1 -23202.118,E2 -23202.118} C_VEL
LIN {X 0,Y 164.635,Z 379.554,A -85,B 0,C 180,E1 -23207.677,E2 -23207.677} C_VEL
LIN {X 0,Y 164.794,Z 379.531,A -85,B 0,C 180,E1 -23210.179,E2 -23210.179} C_VEL
LIN {X 0,Y 164.844,Z 379.56,A -85,B 0,C 180,E1 -23212.652,E2 -23212.652} C_VEL
LIN {X 0,Y 165.048,Z 379.523,A -85,B 0,C 180,E1 -23217.56,E2 -23217.56} C_VEL
LIN {X 0,Y 165.294,Z 379.496,A -85,B 0,C 180,E1 -23220.001,E2 -23220.001} C_VEL
LIN {X 0,Y 164.772,Z 379.567,A -85,B 0,C 180,E1 -23224.895,E2 -23224.895} C_VEL
LIN {X 0,Y 164.857,Z 379.54,A -85,B 0,C 180,E1 -23227.349,E2 -23227.349} C_VEL
LIN {X 0,Y 164.778,Z 379.584,A -85,B 0,C 180,E1 -23231.198,E2 -23231.198} C_VEL
LIN {X 0,Y 164.482,Z 379.588,A -85,B 0,C 180,E1 -23237.404,E2 -23237.404} C_VEL
LIN {X 0,Y 164.472,Z 379.619,A -85,B 0,C 180,E1 -23239.99,E2 -23239.99} C_VEL
LIN {X 0,Y 164.385,Z 379.596,A -85,B 0,C 180,E1 -23246.13,E2 -23246.13} C_VEL
LIN {X 0,Y 164.388,Z 379.631,A -85,B 0,C 180,E1 -23251.237,E2 -23251.237} C_VEL
LIN {X 0,Y 164.294,Z 379.621,A -85,B 0,C 180,E1 -23256.791,E2 -23256.791} C_VEL
LIN {X 0,Y 164.29,Z 379.645,A -85,B 0,C 180,E1 -23259.918,E2 -23259.918} C_VEL
LIN {X 0,Y 164.279,Z 379.616,A -85,B 0,C 180,E1 -23263.343,E2 -23263.343} C_VEL
LIN {X 0,Y 164.264,Z 379.647,A -85,B 0,C 180,E1 -23266.801,E2 -23266.801} C_VEL
LIN {X 0,Y 164.292,Z 379.622,A -85,B 0,C 180,E1 -23270.355,E2 -23270.355} C_VEL
LIN {X 0,Y 164.327,Z 379.641,A -85,B 0,C 180,E1 -23274.352,E2 -23274.352} C_VEL
LIN {X 0,Y 164.377,Z 379.616,A -85,B 0,C 180,E1 -23279.013,E2 -23279.013} C_VEL
LIN {X 0,Y 165.202,Z 382.184,A -85,B 0,C 180,E1 -23279.723,E2 -23279.723} C_VEL
LIN {X 0,Y 167.159,Z 384.442,A -85,B 0,C 180,E1 -23280.977,E2 -23280.977} C_VEL
LIN {X 0,Y 168.371,Z 385.435,A -85,B 0,C 180,E1 -23281.683,E2 -23281.683} C_VEL
LIN {X 0,Y 170.239,Z 388.48,A -85,B 0,C 180,E1 -23282.87,E2 -23282.87} C_VEL
LIN {X 0,Y 172.347,Z 390.711,A -85,B 0,C 180,E1 -23284.066,E2 -23284.066} C_VEL
LIN {X 0,Y 174.941,Z 394.355,A -85,B 0,C 180,E1 -23285.526,E2 -23285.526} C_VEL
LIN {X 0,Y 176.301,Z 396.19,A -85,B 0,C 180,E1 -23286.25,E2 -23286.25} C_VEL
LIN {X 0,Y 179.911,Z 401.099,A -85,B 0,C 180,E1 -23288.082,E2 -23288.082} C_VEL
LIN {X 0,Y 185.218,Z 408.774,A -85,B 0,C 180,E1 -23290.627,E2 -23290.627} C_VEL
LIN {X 0,Y 193.116,Z 420.649,A -85,B 0,C 180,E1 -23294.014,E2 -23294.014} C_VEL
LIN {X 0,Y 198.498,Z 430.068,A -85,B 0,C 180,E1 -23296.183,E2 -23296.183} C_VEL
LIN {X 0,Y 204.929,Z 441.373,A -85,B 0,C 180,E1 -23298.559,E2 -23298.559} C_VEL
LIN {X 0,Y 209.647,Z 451.33,A -85,B 0,C 180,E1 -23300.268,E2 -23300.268} C_VEL
LIN {X 0,Y 209.82,Z 452.284,A -85,B 0,C 180,E1 -23300.36,E2 -23300.36} C_VEL
LIN {X 0,Y 203.908,Z 526.578,A -85,B 0,C 180,E1 -23302.948,E2 -23302.948} C_VEL
LIN {X 0,Y 202.039,Z 541.142,A -85,B 0,C 180,E1 -23303.76,E2 -23303.76} C_VEL
LIN {X 0,Y 199.488,Z 556.058,A -85,B 0,C 180,E1 -23304.948,E2 -23304.948} C_VEL
LIN {X 0,Y 196.082,Z 571.294,A -85,B 0,C 180,E1 -23306.562,E2 -23306.562} C_VEL
LIN {X 0,Y 192.462,Z 584.909,A -85,B 0,C 180,E1 -23308.432,E2 -23308.432} C_VEL
LIN {X 0,Y 188.188,Z 598.575,A -85,B 0,C 180,E1 -23310.803,E2 -23310.803} C_VEL
LIN {X 0,Y 183.679,Z 611.367,A -85,B 0,C 180,E1 -23313.61,E2 -23313.61} C_VEL
LIN {X 0,Y 179.311,Z 622.791,A -85,B 0,C 180,E1 -23316.754,E2 -23316.754} C_VEL
LIN {X 0,Y 175.678,Z 631.803,A -85,B 0,C 180,E1 -23319.79,E2 -23319.79} C_VEL
LIN {X 0,Y 172.107,Z 640.357,A -85,B 0,C 180,E1 -23323.325,E2 -23323.325} C_VEL
LIN {X 0,Y 168.684,Z 648.665,A -85,B 0,C 180,E1 -23327.581,E2 -23327.581} C_VEL
LIN {X 0,Y 165.768,Z 656.093,A -85,B 0,C 180,E1 -23332.432,E2 -23332.432} C_VEL
LIN {X 0,Y 163.875,Z 661.496,A -85,B 0,C 180,E1 -23337.019,E2 -23337.019} C_VEL
LIN {X 0,Y 162.623,Z 665.349,A -85,B 0,C 180,E1 -23341.24,E2 -23341.24} C_VEL
LIN {X 0,Y 161.996,Z 667.638,A -85,B 0,C 180,E1 -23344.481,E2 -23344.481} C_VEL
LIN {X 0,Y 161.743,Z 669.807,A -85,B 0,C 180,E1 -23348.542,E2 -23348.542} C_VEL
LIN {X 0,Y 162.056,Z 671.44,A -85,B 0,C 180,E1 -23353.94,E2 -23353.94} C_VEL
LIN {X 0,Y 163.285,Z 671.729,A -85,B 0,C 180,E1 -23359.787,E2 -23359.787} C_VEL
LIN {X 0,Y 164.951,Z 670.912,A -85,B 0,C 180,E1 -23364.051,E2 -23364.051} C_VEL
LIN {X 0,Y 166.792,Z 669.681,A -85,B 0,C 180,E1 -23367.431,E2 -23367.431} C_VEL
LIN {X 0,Y 169.114,Z 667.849,A -85,B 0,C 180,E1 -23370.777,E2 -23370.777} C_VEL
LIN {X 0,Y 171.939,Z 665.376,A -85,B 0,C 180,E1 -23374.062,E2 -23374.062} C_VEL
LIN {X 0,Y 176.397,Z 661.226,A -85,B 0,C 180,E1 -23378.2,E2 -23378.2} C_VEL
LIN {X 0,Y 181.308,Z 656.212,A -85,B 0,C 180,E1 -23381.934,E2 -23381.934} C_VEL
LIN {X 0,Y 188.213,Z 648.661,A -85,B 0,C 180,E1 -23386.138,E2 -23386.138} C_VEL
LIN {X 0,Y 195.111,Z 640.326,A -85,B 0,C 180,E1 -23389.623,E2 -23389.623} C_VEL
LIN {X 0,Y 201.553,Z 631.632,A -85,B 0,C 180,E1 -23392.469,E2 -23392.469} C_VEL
LIN {X 0,Y 208.692,Z 621.06,A -85,B 0,C 180,E1 -23395.171,E2 -23395.171} C_VEL
LIN {X 0,Y 215.457,Z 609.787,A -85,B 0,C 180,E1 -23397.429,E2 -23397.429} C_VEL
LIN {X 0,Y 221.663,Z 597.912,A -85,B 0,C 180,E1 -23399.318,E2 -23399.318} C_VEL
LIN {X 0,Y 227.092,Z 585.758,A -85,B 0,C 180,E1 -23400.887,E2 -23400.887} C_VEL
LIN {X 0,Y 232.47,Z 571.557,A -85,B 0,C 180,E1 -23402.311,E2 -23402.311} C_VEL
LIN {X 0,Y 236.701,Z 557.721,A -85,B 0,C 180,E1 -23403.404,E2 -23403.404} C_VEL
LIN {X 0,Y 240.298,Z 542.594,A -85,B 0,C 180,E1 -23404.282,E2 -23404.282} C_VEL
LIN {X 0,Y 242.811,Z 527.599,A -85,B 0,C 180,E1 -23404.895,E2 -23404.895} C_VEL
LIN {X 0,Y 248.912,Z 475.393,A -85,B 0,C 180,E1 -23406.429,E2 -23406.429} C_VEL
LIN {X 0,Y 246.965,Z 470.276,A -85,B 0,C 180,E1 -23408.535,E2 -23408.535} C_VEL
LIN {X 0,Y 244.885,Z 466.206,A -85,B 0,C 180,E1 -23411.14,E2 -23411.14} C_VEL
LIN {X 0,Y 243.588,Z 463.429,A -85,B 0,C 180,E1 -23413.345,E2 -23413.345} C_VEL
LIN {X 0,Y 242.196,Z 460.559,A -85,B 0,C 180,E1 -23417.821,E2 -23417.821} C_VEL
LIN {X 0,Y 242.142,Z 460.135,A -85,B 0,C 180,E1 -23418.618,E2 -23418.618} C_VEL
LIN {X 0,Y 242.27,Z 461.635,A -85,B 0,C 180,E1 -23422.416,E2 -23422.416} C_VEL
LIN {X 0,Y 243.652,Z 466.391,A -85,B 0,C 180,E1 -23426.521,E2 -23426.521} C_VEL
LIN {X 0,Y 245.078,Z 471.065,A -85,B 0,C 180,E1 -23429.022,E2 -23429.022} C_VEL
LIN {X 0,Y 246.86,Z 476.766,A -85,B 0,C 180,E1 -23431.34,E2 -23431.34} C_VEL
LIN {X 0,Y 248.383,Z 482.412,A -85,B 0,C 180,E1 -23433.093,E2 -23433.093} C_VEL
LIN {X 0,Y 241.381,Z 540.857,A -85,B 0,C 180,E1 -23434.751,E2 -23434.751} C_VEL
LIN {X 0,Y 238.192,Z 557.026,A -85,B 0,C 180,E1 -23435.402,E2 -23435.402} C_VEL
LIN {X 0,Y 234.056,Z 572.017,A -85,B 0,C 180,E1 -23436.197,E2 -23436.197} C_VEL
LIN {X 0,Y 230.472,Z 582.682,A -85,B 0,C 180,E1 -23436.952,E2 -23436.952} C_VEL
LIN {X 0,Y 228.226,Z 588.02,A -85,B 0,C 180,E1 -23437.248,E2 -23437.248} C_VEL
LIN {X 0,Y 223.368,Z 596.624,A -85,B 0,C 180,E1 -23437.391,E2 -23437.391} C_VEL
LIN {X 0,Y 218.14,Z 605.029,A -85,B 0,C 180,E1 -23437.604,E2 -23437.604} C_VEL
LIN {X 0,Y 215.291,Z 609.888,A -85,B 0,C 180,E1 -23438.029,E2 -23438.029} C_VEL
LIN {X 0,Y 207.864,Z 623.125,A -85,B 0,C 180,E1 -23440.006,E2 -23440.006} C_VEL
LIN {X 0,Y 201.05,Z 633.77,A -85,B 0,C 180,E1 -23442.026,E2 -23442.026} C_VEL
LIN {X 0,Y 194.199,Z 643.516,A -85,B 0,C 180,E1 -23444.376,E2 -23444.376} C_VEL
LIN {X 0,Y 186.824,Z 653.184,A -85,B 0,C 180,E1 -23447.379,E2 -23447.379} C_VEL
LIN {X 0,Y 179.985,Z 661.409,A -85,B 0,C 180,E1 -23450.614,E2 -23450.614} C_VEL
LIN {X 0,Y 173.235,Z 669.027,A -85,B 0,C 180,E1 -23454.553,E2 -23454.553} C_VEL
LIN {X 0,Y 167.938,Z 674.771,A -85,B 0,C 180,E1 -23458.458,E2 -23458.458} C_VEL
LIN {X 0,Y 162.963,Z 679.982,A -85,B 0,C 180,E1 -23463.074,E2 -23463.074} C_VEL
LIN {X 0,Y 159.149,Z 684.02,A -85,B 0,C 180,E1 -23468.025,E2 -23468.025} C_VEL
LIN {X 0,Y 156.168,Z 687.318,A -85,B 0,C 180,E1 -23474.334,E2 -23474.334} C_VEL
LIN {X 0,Y 155.059,Z 688.78,A -85,B 0,C 180,E1 -23479.553,E2 -23479.553} C_VEL
LIN {X 0,Y 154.944,Z 689.093,A -85,B 0,C 180,E1 -23484.794,E2 -23484.794} C_VEL
LIN {X 0,Y 155.132,Z 688.808,A -85,B 0,C 180,E1 -23487.402,E2 -23487.402} C_VEL
LIN {X 0,Y 155.316,Z 688.222,A -85,B 0,C 180,E1 -23489.999,E2 -23489.999} C_VEL
LIN {X 0,Y 155.101,Z 686.403,A -85,B 0,C 180,E1 -23494.541,E2 -23494.541} C_VEL
LIN {X 0,Y 154.996,Z 684.446,A -85,B 0,C 180,E1 -23497.817,E2 -23497.817} C_VEL
LIN {X 0,Y 155.571,Z 680.241,A -85,B 0,C 180,E1 -23503.053,E2 -23503.053} C_VEL
LIN {X 0,Y 157.086,Z 674.563,A -85,B 0,C 180,E1 -23508.25,E2 -23508.25} C_VEL
LIN {X 0,Y 159.721,Z 667.273,A -85,B 0,C 180,E1 -23513.328,E2 -23513.328} C_VEL
LIN {X 0,Y 162.918,Z 659.414,A -85,B 0,C 180,E1 -23517.627,E2 -23517.627} C_VEL
LIN {X 0,Y 166.269,Z 651.392,A -85,B 0,C 180,E1 -23521.183,E2 -23521.183} C_VEL
LIN {X 0,Y 170.98,Z 640.198,A -85,B 0,C 180,E1 -23525.13,E2 -23525.13} C_VEL
LIN {X 0,Y 175.671,Z 628.67,A -85,B 0,C 180,E1 -23528.322,E2 -23528.322} C_VEL
LIN {X 0,Y 180.513,Z 616.033,A -85,B 0,C 180,E1 -23531.07,E2 -23531.07} C_VEL
LIN {X 0,Y 184.779,Z 603.659,A -85,B 0,C 180,E1 -23533.204,E2 -23533.204} C_VEL
LIN {X 0,Y 188.661,Z 590.268,A -85,B 0,C 180,E1 -23535.054,E2 -23535.054} C_VEL
LIN {X 0,Y 192.333,Z 575.785,A -85,B 0,C 180,E1 -23536.571,E2 -23536.571} C_VEL
LIN {X 0,Y 195.114,Z 561.68,A -85,B 0,C 180,E1 -23537.69,E2 -23537.69} C_VEL
LIN {X 0,Y 197.531,Z 546.125,A -85,B 0,C 180,E1 -23538.536,E2 -23538.536} C_VEL
LIN {X 0,Y 201.617,Z 497.573,A -85,B 0,C 180,E1 -23540.285,E2 -23540.285} C_VEL
LIN {X 0,Y 204.179,Z 465.528,A -85,B 0,C 180,E1 -23541.401,E2 -23541.401} C_VEL
LIN {X 0,Y 197.758,Z 449.135,A -85,B 0,C 180,E1 -23544.021,E2 -23544.021} C_VEL
LIN {X 0,Y 190.905,Z 433.838,A -85,B 0,C 180,E1 -23546.955,E2 -23546.955} C_VEL
LIN {X 0,Y 184.381,Z 420.631,A -85,B 0,C 180,E1 -23549.982,E2 -23549.982} C_VEL
LIN {X 0,Y 177.775,Z 408.553,A -85,B 0,C 180,E1 -23553.337,E2 -23553.337} C_VEL
LIN {X 0,Y 174.472,Z 403.772,A -85,B 0,C 180,E1 -23555.059,E2 -23555.059} C_VEL
LIN {X 0,Y 171.671,Z 399.979,A -85,B 0,C 180,E1 -23556.595,E2 -23556.595} C_VEL
LIN {X 0,Y 168.554,Z 395.647,A -85,B 0,C 180,E1 -23558.443,E2 -23558.443} C_VEL
LIN {X 0,Y 166.044,Z 392.389,A -85,B 0,C 180,E1 -23560.027,E2 -23560.027} C_VEL
LIN {X 0,Y 165.236,Z 391.079,A -85,B 0,C 180,E1 -23560.574,E2 -23560.574} C_VEL
LIN {X 0,Y 162.749,Z 388.382,A -85,B 0,C 180,E1 -23562.193,E2 -23562.193} C_VEL
LIN {X 0,Y 161.414,Z 385.987,A -85,B 0,C 180,E1 -23563.202,E2 -23563.202} C_VEL
LIN {X 0,Y 159.104,Z 384.17,A -85,B 0,C 180,E1 -23564.796,E2 -23564.796} C_VEL
LIN {X 0,Y 157.796,Z 381.818,A -85,B 0,C 180,E1 -23565.904,E2 -23565.904} C_VEL
LIN {X 0,Y 157.502,Z 380.458,A -85,B 0,C 180,E1 -23566.288,E2 -23566.288} C_VEL
LIN {X 0,Y 157.722,Z 380.408,A -85,B 0,C 180,E1 -23569.734,E2 -23569.734} C_VEL
LIN {X 0,Y 157.782,Z 380.43,A -85,B 0,C 180,E1 -23572.322,E2 -23572.322} C_VEL
LIN {X 0,Y 158.256,Z 380.371,A -85,B 0,C 180,E1 -23580.001,E2 -23580.001} C_VEL
LIN {X 0,Y 157.82,Z 380.416,A -85,B 0,C 180,E1 -23587.678,E2 -23587.678} C_VEL
LIN {X 0,Y 157.703,Z 380.466,A -85,B 0,C 180,E1 -23591.361,E2 -23591.361} C_VEL
LIN {X 0,Y 157.459,Z 380.461,A -85,B 0,C 180,E1 -23595.535,E2 -23595.535} C_VEL
LIN {X 0,Y 157.366,Z 380.508,A -85,B 0,C 180,E1 -23600.934,E2 -23600.934} C_VEL
LIN {X 0,Y 157.308,Z 380.479,A -85,B 0,C 180,E1 -23606.682,E2 -23606.682} C_VEL
LIN {X 0,Y 157.281,Z 380.502,A -85,B 0,C 180,E1 -23612.427,E2 -23612.427} C_VEL
LIN {X 0,Y 157.267,Z 380.491,A -85,B 0,C 180,E1 -23616.451,E2 -23616.451} C_VEL
LIN {X 0,Y 157.192,Z 380.503,A -85,B 0,C 180,E1 -23622.118,E2 -23622.118} C_VEL
LIN {X 0,Y 157.192,Z 380.531,A -85,B 0,C 180,E1 -23627.885,E2 -23627.885} C_VEL
LIN {X 0,Y 157.261,Z 380.509,A -85,B 0,C 180,E1 -23633.556,E2 -23633.556} C_VEL
LIN {X 0,Y 157.281,Z 380.631,A -85,B 0,C 180,E1 -23634.757,E2 -23634.757} C_VEL
LIN {X 0,Y 158.109,Z 383.084,A -85,B 0,C 180,E1 -23635.576,E2 -23635.576} C_VEL
LIN {X 0,Y 160.124,Z 385.372,A -85,B 0,C 180,E1 -23637.081,E2 -23637.081} C_VEL
LIN {X 0,Y 161.646,Z 386.506,A -85,B 0,C 180,E1 -23638.126,E2 -23638.126} C_VEL
LIN {X 0,Y 163.424,Z 389.504,A -85,B 0,C 180,E1 -23639.449,E2 -23639.449} C_VEL
LIN {X 0,Y 165.606,Z 391.726,A -85,B 0,C 180,E1 -23640.839,E2 -23640.839} C_VEL
LIN {X 0,Y 168.003,Z 395.159,A -85,B 0,C 180,E1 -23642.363,E2 -23642.363} C_VEL
LIN {X 0,Y 169.508,Z 396.863,A -85,B 0,C 180,E1 -23643.248,E2 -23643.248} C_VEL
LIN {X 0,Y 172.299,Z 400.64,A -85,B 0,C 180,E1 -23644.873,E2 -23644.873} C_VEL
LIN {X 0,Y 179.228,Z 410.492,A -85,B 0,C 180,E1 -23648.513,E2 -23648.513} C_VEL
LIN {X 0,Y 186.572,Z 421.651,A -85,B 0,C 180,E1 -23651.967,E2 -23651.967} C_VEL
LIN {X 0,Y 192.303,Z 431.003,A -85,B 0,C 180,E1 -23654.414,E2 -23654.414} C_VEL
LIN {X 0,Y 200.911,Z 446.648,A -85,B 0,C 180,E1 -23657.797,E2 -23657.797} C_VEL
LIN {X 0,Y 204.305,Z 454.017,A -85,B 0,C 180,E1 -23659.097,E2 -23659.097} C_VEL
LIN {X 0,Y 198.416,Z 526.401,A -85,B 0,C 180,E1 -23661.666,E2 -23661.666} C_VEL
LIN {X 0,Y 196.363,Z 541.923,A -85,B 0,C 180,E1 -23662.546,E2 -23662.546} C_VEL
LIN {X 0,Y 193.726,Z 556.735,A -85,B 0,C 180,E1 -23663.753,E2 -23663.753} C_VEL
LIN {X 0,Y 190.398,Z 571.192,A -85,B 0,C 180,E1 -23665.306,E2 -23665.306} C_VEL
LIN {X 0,Y 186.453,Z 585.48,A -85,B 0,C 180,E1 -23667.3,E2 -23667.3} C_VEL
LIN {X 0,Y 182.282,Z 598.409,A -85,B 0,C 180,E1 -23669.579,E2 -23669.579} C_VEL
LIN {X 0,Y 177.89,Z 610.563,A -85,B 0,C 180,E1 -23672.265,E2 -23672.265} C_VEL
LIN {X 0,Y 173.67,Z 621.325,A -85,B 0,C 180,E1 -23675.225,E2 -23675.225} C_VEL
LIN {X 0,Y 169.4,Z 631.448,A -85,B 0,C 180,E1 -23678.654,E2 -23678.654} C_VEL
LIN {X 0,Y 165.524,Z 640.404,A -85,B 0,C 180,E1 -23682.426,E2 -23682.426} C_VEL
LIN {X 0,Y 162.529,Z 647.363,A -85,B 0,C 180,E1 -23686.014,E2 -23686.014} C_VEL
LIN {X 0,Y 159.471,Z 654.612,A -85,B 0,C 180,E1 -23690.645,E2 -23690.645} C_VEL
LIN {X 0,Y 157.471,Z 660.007,A -85,B 0,C 180,E1 -23694.997,E2 -23694.997} C_VEL
LIN {X 0,Y 155.902,Z 664.534,A -85,B 0,C 180,E1 -23699.729,E2 -23699.729} C_VEL
LIN {X 0,Y 154.816,Z 668.372,A -85,B 0,C 180,E1 -23705.2,E2 -23705.2} C_VEL
LIN {X 0,Y 154.639,Z 670.444,A -85,B 0,C 180,E1 -23709.516,E2 -23709.516} C_VEL
LIN {X 0,Y 154.887,Z 671.616,A -85,B 0,C 180,E1 -23713.446,E2 -23713.446} C_VEL
LIN {X 0,Y 155.532,Z 672.19,A -85,B 0,C 180,E1 -23717.326,E2 -23717.326} C_VEL
LIN {X 0,Y 157.516,Z 671.794,A -85,B 0,C 180,E1 -23723.431,E2 -23723.431} C_VEL
LIN {X 0,Y 160.065,Z 670.311,A -85,B 0,C 180,E1 -23728.204,E2 -23728.204} C_VEL
LIN {X 0,Y 162.467,Z 668.64,A -85,B 0,C 180,E1 -23731.585,E2 -23731.585} C_VEL
LIN {X 0,Y 167.726,Z 664.365,A -85,B 0,C 180,E1 -23737.198,E2 -23737.198} C_VEL
LIN {X 0,Y 172.292,Z 660.246,A -85,B 0,C 180,E1 -23740.953,E2 -23740.953} C_VEL
LIN {X 0,Y 178.644,Z 654.07,A -85,B 0,C 180,E1 -23745.184,E2 -23745.184} C_VEL
LIN {X 0,Y 184.611,Z 647.742,A -85,B 0,C 180,E1 -23748.47,E2 -23748.47} C_VEL
LIN {X 0,Y 191.713,Z 639.458,A -85,B 0,C 180,E1 -23751.813,E2 -23751.813} C_VEL
LIN {X 0,Y 199.24,Z 629.714,A -85,B 0,C 180,E1 -23754.86,E2 -23754.86} C_VEL
LIN {X 0,Y 206.356,Z 619.397,A -85,B 0,C 180,E1 -23757.354,E2 -23757.354} C_VEL
LIN {X 0,Y 212.883,Z 608.714,A -85,B 0,C 180,E1 -23759.394,E2 -23759.394} C_VEL
LIN {X 0,Y 220.111,Z 595.021,A -85,B 0,C 180,E1 -23761.452,E2 -23761.452} C_VEL
LIN {X 0,Y 225.584,Z 582.837,A -85,B 0,C 180,E1 -23762.912,E2 -23762.912} C_VEL
LIN {X 0,Y 231.038,Z 568.22,A -85,B 0,C 180,E1 -23764.254,E2 -23764.254} C_VEL
LIN {X 0,Y 235.109,Z 554.459,A -85,B 0,C 180,E1 -23765.252,E2 -23765.252} C_VEL
LIN {X 0,Y 238.53,Z 539.318,A -85,B 0,C 180,E1 -23766.052,E2 -23766.052} C_VEL
LIN {X 0,Y 241.041,Z 523.118,A -85,B 0,C 180,E1 -23766.618,E2 -23766.618} C_VEL
LIN {X 0,Y 246.328,Z 479.598,A -85,B 0,C 180,E1 -23767.861,E2 -23767.861} C_VEL
LIN {X 0,Y 245.084,Z 476.29,A -85,B 0,C 180,E1 -23769.341,E2 -23769.341} C_VEL
LIN {X 0,Y 243.413,Z 472.821,A -85,B 0,C 180,E1 -23771.66,E2 -23771.66} C_VEL
LIN {X 0,Y 242.235,Z 470.248,A -85,B 0,C 180,E1 -23773.862,E2 -23773.862} C_VEL
LIN {X 0,Y 241.058,Z 467.176,A -85,B 0,C 180,E1 -23778.705,E2 -23778.705} C_VEL
LIN {X 0,Y 241.142,Z 468.587,A -85,B 0,C 180,E1 -23782.139,E2 -23782.139} C_VEL
LIN {X 0,Y 242.25,Z 473.056,A -85,B 0,C 180,E1 -23786.015,E2 -23786.015} C_VEL
LIN {X 0,Y 243.499,Z 477.447,A -85,B 0,C 180,E1 -23788.389,E2 -23788.389} C_VEL
LIN {X 0,Y 244.926,Z 482.597,A -85,B 0,C 180,E1 -23790.505,E2 -23790.505} C_VEL
LIN {X 0,Y 245.752,Z 486.049,A -85,B 0,C 180,E1 -23791.621,E2 -23791.621} C_VEL
LIN {X 0,Y 239.035,Z 540.067,A -85,B 0,C 180,E1 -23793.136,E2 -23793.136} C_VEL
LIN {X 0,Y 235.91,Z 555.842,A -85,B 0,C 180,E1 -23793.761,E2 -23793.761} C_VEL
LIN {X 0,Y 231.834,Z 570.485,A -85,B 0,C 180,E1 -23794.493,E2 -23794.493} C_VEL
LIN {X 0,Y 227.283,Z 583.536,A -85,B 0,C 180,E1 -23795.381,E2 -23795.381} C_VEL
LIN {X 0,Y 221.208,Z 597.968,A -85,B 0,C 180,E1 -23796.656,E2 -23796.656} C_VEL
LIN {X 0,Y 215.291,Z 609.888,A -85,B 0,C 180,E1 -23798.029,E2 -23798.029} C_VEL
LIN {X 0,Y 212.346,Z 614.729,A -85,B 0,C 180,E1 -23798.509,E2 -23798.509} C_VEL
LIN {X 0,Y 206.411,Z 622.504,A -85,B 0,C 180,E1 -23799.005,E2 -23799.005} C_VEL
LIN {X 0,Y 200.282,Z 629.919,A -85,B 0,C 180,E1 -23799.632,E2 -23799.632} C_VEL
LIN {X 0,Y 197.017,Z 634.122,A -85,B 0,C 180,E1 -23800.336,E2 -23800.336} C_VEL
LIN {X 0,Y 189.346,Z 644.435,A -85,B 0,C 180,E1 -23802.855,E2 -23802.855} C_VEL
LIN {X 0,Y 181.7,Z 653.864,A -85,B 0,C 180,E1 -23805.874,E2 -23805.874} C_VEL
LIN {X 0,Y 174.549,Z 661.857,A -85,B 0,C 180,E1 -23809.133,E2 -23809.133} C_VEL
LIN {X 0,Y 168.207,Z 668.607,A -85,B 0,C 180,E1 -23812.706,E2 -23812.706} C_VEL
LIN {X 0,Y 161.899,Z 674.944,A -85,B 0,C 180,E1 -23817.136,E2 -23817.136} C_VEL
LIN {X 0,Y 156.598,Z 679.974,A -85,B 0,C 180,E1 -23821.884,E2 -23821.884} C_VEL
LIN {X 0,Y 152.315,Z 684.078,A -85,B 0,C 180,E1 -23827.341,E2 -23827.341} C_VEL
LIN {X 0,Y 149.264,Z 687.047,A -85,B 0,C 180,E1 -23833.589,E2 -23833.589} C_VEL
LIN {X 0,Y 148.017,Z 688.386,A -85,B 0,C 180,E1 -23839.05,E2 -23839.05} C_VEL
LIN {X 0,Y 147.842,Z 688.637,A -85,B 0,C 180,E1 -23844.543,E2 -23844.543} C_VEL
LIN {X 0,Y 148.051,Z 688.306,A -85,B 0,C 180,E1 -23847.278,E2 -23847.278} C_VEL
LIN {X 0,Y 148.252,Z 687.665,A -85,B 0,C 180,E1 -23849.999,E2 -23849.999} C_VEL
LIN {X 0,Y 148.021,Z 685.922,A -85,B 0,C 180,E1 -23854.393,E2 -23854.393} C_VEL
LIN {X 0,Y 147.933,Z 683.717,A -85,B 0,C 180,E1 -23858.193,E2 -23858.193} C_VEL
LIN {X 0,Y 148.597,Z 679.391,A -85,B 0,C 180,E1 -23863.677,E2 -23863.677} C_VEL
LIN {X 0,Y 150.278,Z 673.585,A -85,B 0,C 180,E1 -23869.108,E2 -23869.108} C_VEL
LIN {X 0,Y 153.112,Z 666.153,A -85,B 0,C 180,E1 -23874.399,E2 -23874.399} C_VEL
LIN {X 0,Y 156.588,Z 658.15,A -85,B 0,C 180,E1 -23878.846,E2 -23878.846} C_VEL
LIN {X 0,Y 160.784,Z 648.446,A -85,B 0,C 180,E1 -23883.118,E2 -23883.118} C_VEL
LIN {X 0,Y 165.136,Z 638.552,A -85,B 0,C 180,E1 -23886.57,E2 -23886.57} C_VEL
LIN {X 0,Y 170.059,Z 626.781,A -85,B 0,C 180,E1 -23889.833,E2 -23889.833} C_VEL
LIN {X 0,Y 175.138,Z 613.857,A -85,B 0,C 180,E1 -23892.621,E2 -23892.621} C_VEL
LIN {X 0,Y 179.845,Z 600.101,A -85,B 0,C 180,E1 -23894.946,E2 -23894.946} C_VEL
LIN {X 0,Y 184.194,Z 585.318,A -85,B 0,C 180,E1 -23896.861,E2 -23896.861} C_VEL
LIN {X 0,Y 187.79,Z 570.837,A -85,B 0,C 180,E1 -23898.257,E2 -23898.257} C_VEL
LIN {X 0,Y 190.537,Z 556.078,A -85,B 0,C 180,E1 -23899.326,E2 -23899.326} C_VEL
LIN {X 0,Y 192.473,Z 541.431,A -85,B 0,C 180,E1 -23900.066,E2 -23900.066} C_VEL
LIN {X 0,Y 198.805,Z 467.723,A -85,B 0,C 180,E1 -23902.668,E2 -23902.668} C_VEL
LIN {X 0,Y 192.665,Z 452.035,A -85,B 0,C 180,E1 -23905.283,E2 -23905.283} C_VEL
LIN {X 0,Y 186.301,Z 437.548,A -85,B 0,C 180,E1 -23908.201,E2 -23908.201} C_VEL
LIN {X 0,Y 180.163,Z 424.94,A -85,B 0,C 180,E1 -23911.195,E2 -23911.195} C_VEL
LIN {X 0,Y 174.239,Z 413.872,A -85,B 0,C 180,E1 -23914.364,E2 -23914.364} C_VEL
LIN {X 0,Y 169.36,Z 406.599,A -85,B 0,C 180,E1 -23917.106,E2 -23917.106} C_VEL
LIN {X 0,Y 166.232,Z 402.26,A -85,B 0,C 180,E1 -23919.021,E2 -23919.021} C_VEL
LIN {X 0,Y 163.011,Z 398.024,A -85,B 0,C 180,E1 -23921.103,E2 -23921.103} C_VEL
LIN {X 0,Y 159.463,Z 393.428,A -85,B 0,C 180,E1 -23923.601,E2 -23923.601} C_VEL
LIN {X 0,Y 158.604,Z 392.212,A -85,B 0,C 180,E1 -23924.253,E2 -23924.253} C_VEL
LIN {X 0,Y 156.2,Z 389.708,A -85,B 0,C 180,E1 -23926.089,E2 -23926.089} C_VEL
LIN {X 0,Y 154.684,Z 386.924,A -85,B 0,C 180,E1 -23927.477,E2 -23927.477} C_VEL
LIN {X 0,Y 152.258,Z 384.933,A -85,B 0,C 180,E1 -23929.529,E2 -23929.529} C_VEL
LIN {X 0,Y 151.012,Z 382.754,A -85,B 0,C 180,E1 -23930.795,E2 -23930.795} C_VEL
LIN {X 0,Y 150.678,Z 381.296,A -85,B 0,C 180,E1 -23931.282,E2 -23931.282} C_VEL
LIN {X 0,Y 150.897,Z 381.284,A -85,B 0,C 180,E1 -23937.331,E2 -23937.331} C_VEL
LIN {X 0,Y 151.216,Z 381.246,A -85,B 0,C 180,E1 -23940.001,E2 -23940.001} C_VEL
LIN {X 0,Y 150.759,Z 381.296,A -85,B 0,C 180,E1 -23948.04,E2 -23948.04} C_VEL
LIN {X 0,Y 150.632,Z 381.347,A -85,B 0,C 180,E1 -23951.545,E2 -23951.545} C_VEL
LIN {X 0,Y 150.364,Z 381.341,A -85,B 0,C 180,E1 -23956.287,E2 -23956.287} C_VEL
LIN {X 0,Y 150.348,Z 381.382,A -85,B 0,C 180,E1 -23960.792,E2 -23960.792} C_VEL
LIN {X 0,Y 150.241,Z 381.362,A -85,B 0,C 180,E1 -23967.282,E2 -23967.282} C_VEL
LIN {X 0,Y 150.219,Z 381.376,A -85,B 0,C 180,E1 -23972.637,E2 -23972.637} C_VEL
LIN {X 0,Y 150.177,Z 381.384,A -85,B 0,C 180,E1 -23977.474,E2 -23977.474} C_VEL
LIN {X 0,Y 150.135,Z 381.387,A -85,B 0,C 180,E1 -23981.5,E2 -23981.5} C_VEL
LIN {X 0,Y 150.125,Z 381.387,A -85,B 0,C 180,E1 -23985.397,E2 -23985.397} C_VEL
LIN {X 0,Y 150.164,Z 381.443,A -85,B 0,C 180,E1 -23989.466,E2 -23989.466} C_VEL
LIN {X 0,Y 150.899,Z 383.816,A -85,B 0,C 180,E1 -23990.39,E2 -23990.39} C_VEL
LIN {X 0,Y 152.832,Z 386.078,A -85,B 0,C 180,E1 -23992.223,E2 -23992.223} C_VEL
LIN {X 0,Y 154.706,Z 387.235,A -85,B 0,C 180,E1 -23993.745,E2 -23993.745} C_VEL
LIN {X 0,Y 156.322,Z 390.252,A -85,B 0,C 180,E1 -23995.202,E2 -23995.202} C_VEL
LIN {X 0,Y 159.127,Z 392.967,A -85,B 0,C 180,E1 -23997.272,E2 -23997.272} C_VEL
LIN {X 0,Y 161.473,Z 396.384,A -85,B 0,C 180,E1 -23999.027,E2 -23999.027} C_VEL
LIN {X 0,Y 162.916,Z 398.02,A -85,B 0,C 180,E1 -23999.997,E2 -23999.997} C_VEL
LIN {X 0,Y 165.832,Z 401.831,A -85,B 0,C 180,E1 -24001.88,E2 -24001.88} C_VEL
LIN {X 0,Y 170.431,Z 408.355,A -85,B 0,C 180,E1 -24004.668,E2 -24004.668} C_VEL
LIN {X 0,Y 175.331,Z 415.245,A -85,B 0,C 180,E1 -24007.33,E2 -24007.33} C_VEL
LIN {X 0,Y 183.552,Z 428.014,A -85,B 0,C 180,E1 -24011.367,E2 -24011.367} C_VEL
LIN {X 0,Y 188.79,Z 436.988,A -85,B 0,C 180,E1 -24013.689,E2 -24013.689} C_VEL
LIN {X 0,Y 196.423,Z 451.022,A -85,B 0,C 180,E1 -24016.836,E2 -24016.836} C_VEL
LIN {X 0,Y 198.95,Z 456.467,A -85,B 0,C 180,E1 -24017.836,E2 -24017.836} C_VEL
LIN {X 0,Y 192.875,Z 527.331,A -85,B 0,C 180,E1 -24020.382,E2 -24020.382} C_VEL
LIN {X 0,Y 190.681,Z 543.027,A -85,B 0,C 180,E1 -24021.3,E2 -24021.3} C_VEL
LIN {X 0,Y 187.777,Z 558.471,A -85,B 0,C 180,E1 -24022.609,E2 -24022.609} C_VEL
LIN {X 0,Y 184.308,Z 572.737,A -85,B 0,C 180,E1 -24024.201,E2 -24024.201} C_VEL
LIN {X 0,Y 180.509,Z 585.946,A -85,B 0,C 180,E1 -24026.094,E2 -24026.094} C_VEL
LIN {X 0,Y 176.194,Z 598.857,A -85,B 0,C 180,E1 -24028.422,E2 -24028.422} C_VEL
LIN {X 0,Y 171.632,Z 611.004,A -85,B 0,C 180,E1 -24031.174,E2 -24031.174} C_VEL
LIN {X 0,Y 167.099,Z 622.133,A -85,B 0,C 180,E1 -24034.333,E2 -24034.333} C_VEL
LIN {X 0,Y 162.512,Z 632.557,A -85,B 0,C 180,E1 -24038.018,E2 -24038.018} C_VEL
LIN {X 0,Y 158.234,Z 642.082,A -85,B 0,C 180,E1 -24042.271,E2 -24042.271} C_VEL
LIN {X 0,Y 154.427,Z 650.591,A -85,B 0,C 180,E1 -24047.111,E2 -24047.111} C_VEL
LIN {X 0,Y 151.582,Z 657.277,A -85,B 0,C 180,E1 -24051.981,E2 -24051.981} C_VEL
LIN {X 0,Y 149.646,Z 662.443,A -85,B 0,C 180,E1 -24056.831,E2 -24056.831} C_VEL
LIN {X 0,Y 148.327,Z 666.28,A -85,B 0,C 180,E1 -24061.472,E2 -24061.472} C_VEL
LIN {X 0,Y 147.66,Z 669.103,A -85,B 0,C 180,E1 -24065.987,E2 -24065.987} C_VEL
LIN {X 0,Y 147.641,Z 671.479,A -85,B 0,C 180,E1 -24071.793,E2 -24071.793} C_VEL
LIN {X 0,Y 148.061,Z 672.333,A -85,B 0,C 180,E1 -24075.4,E2 -24075.4} C_VEL
LIN {X 0,Y 148.831,Z 672.661,A -85,B 0,C 180,E1 -24079.074,E2 -24079.074} C_VEL
LIN {X 0,Y 150.066,Z 672.48,A -85,B 0,C 180,E1 -24082.766,E2 -24082.766} C_VEL
LIN {X 0,Y 151.819,Z 671.785,A -85,B 0,C 180,E1 -24086.437,E2 -24086.437} C_VEL
LIN {X 0,Y 154.052,Z 670.555,A -85,B 0,C 180,E1 -24090.091,E2 -24090.091} C_VEL
LIN {X 0,Y 158.216,Z 667.719,A -85,B 0,C 180,E1 -24095.179,E2 -24095.179} C_VEL
LIN {X 0,Y 163.264,Z 663.813,A -85,B 0,C 180,E1 -24099.855,E2 -24099.855} C_VEL
LIN {X 0,Y 170.032,Z 657.966,A -85,B 0,C 180,E1 -24104.747,E2 -24104.747} C_VEL
LIN {X 0,Y 176.575,Z 651.745,A -85,B 0,C 180,E1 -24108.52,E2 -24108.52} C_VEL
LIN {X 0,Y 184.414,Z 643.553,A -85,B 0,C 180,E1 -24112.253,E2 -24112.253} C_VEL
LIN {X 0,Y 191.823,Z 634.807,A -85,B 0,C 180,E1 -24115.327,E2 -24115.327} C_VEL
LIN {X 0,Y 199.308,Z 624.976,A -85,B 0,C 180,E1 -24117.978,E2 -24117.978} C_VEL
LIN {X 0,Y 206.537,Z 614.365,A -85,B 0,C 180,E1 -24120.22,E2 -24120.22} C_VEL
LIN {X 0,Y 213.282,Z 603.024,A -85,B 0,C 180,E1 -24122.124,E2 -24122.124} C_VEL
LIN {X 0,Y 219.995,Z 589.766,A -85,B 0,C 180,E1 -24123.892,E2 -24123.892} C_VEL
LIN {X 0,Y 225.861,Z 576.008,A -85,B 0,C 180,E1 -24125.29,E2 -24125.29} C_VEL
LIN {X 0,Y 230.846,Z 561.62,A -85,B 0,C 180,E1 -24126.445,E2 -24126.445} C_VEL
LIN {X 0,Y 234.801,Z 546.958,A -85,B 0,C 180,E1 -24127.334,E2 -24127.334} C_VEL
LIN {X 0,Y 237.687,Z 532.413,A -85,B 0,C 180,E1 -24127.954,E2 -24127.954} C_VEL
LIN {X 0,Y 243.896,Z 483.848,A -85,B 0,C 180,E1 -24129.347,E2 -24129.347} C_VEL
LIN {X 0,Y 242.147,Z 479.766,A -85,B 0,C 180,E1 -24131.892,E2 -24131.892} C_VEL
LIN {X 0,Y 241.022,Z 477.127,A -85,B 0,C 180,E1 -24134.144,E2 -24134.144} C_VEL
LIN {X 0,Y 239.972,Z 474.241,A -85,B 0,C 180,E1 -24138.793,E2 -24138.793} C_VEL
LIN {X 0,Y 240.021,Z 475.508,A -85,B 0,C 180,E1 -24141.845,E2 -24141.845} C_VEL
LIN {X 0,Y 240.912,Z 479.689,A -85,B 0,C 180,E1 -24145.493,E2 -24145.493} C_VEL
LIN {X 0,Y 241.953,Z 483.891,A -85,B 0,C 180,E1 -24147.767,E2 -24147.767} C_VEL
LIN {X 0,Y 243.157,Z 488.899,A -85,B 0,C 180,E1 -24149.824,E2 -24149.824} C_VEL
LIN {X 0,Y 243.349,Z 489.798,A -85,B 0,C 180,E1 -24150.118,E2 -24150.118} C_VEL
LIN {X 0,Y 236.887,Z 539.849,A -85,B 0,C 180,E1 -24151.499,E2 -24151.499} C_VEL
LIN {X 0,Y 233.607,Z 555.668,A -85,B 0,C 180,E1 -24152.111,E2 -24152.111} C_VEL
LIN {X 0,Y 229.435,Z 570.124,A -85,B 0,C 180,E1 -24152.81,E2 -24152.81} C_VEL
LIN {X 0,Y 224.124,Z 584.785,A -85,B 0,C 180,E1 -24153.8,E2 -24153.8} C_VEL
LIN {X 0,Y 217.85,Z 598.979,A -85,B 0,C 180,E1 -24155.052,E2 -24155.052} C_VEL
LIN {X 0,Y 211.095,Z 611.956,A -85,B 0,C 180,E1 -24156.562,E2 -24156.562} C_VEL
LIN {X 0,Y 203.654,Z 624.372,A -85,B 0,C 180,E1 -24158.452,E2 -24158.452} C_VEL
LIN {X 0,Y 197.017,Z 634.122,A -85,B 0,C 180,E1 -24160.336,E2 -24160.336} C_VEL
LIN {X 0,Y 193.689,Z 638.276,A -85,B 0,C 180,E1 -24161.103,E2 -24161.103} C_VEL
LIN {X 0,Y 187.027,Z 644.886,A -85,B 0,C 180,E1 -24162.083,E2 -24162.083} C_VEL
LIN {X 0,Y 180.237,Z 651.089,A -85,B 0,C 180,E1 -24163.227,E2 -24163.227} C_VEL
LIN {X 0,Y 176.762,Z 654.506,A -85,B 0,C 180,E1 -24164.262,E2 -24164.262} C_VEL
LIN {X 0,Y 169.251,Z 662.358,A -85,B 0,C 180,E1 -24167.563,E2 -24167.563} C_VEL
LIN {X 0,Y 162.284,Z 669.221,A -85,B 0,C 180,E1 -24171.376,E2 -24171.376} C_VEL
LIN {X 0,Y 155.953,Z 675.122,A -85,B 0,C 180,E1 -24175.714,E2 -24175.714} C_VEL
LIN {X 0,Y 150.323,Z 680.006,A -85,B 0,C 180,E1 -24180.599,E2 -24180.599} C_VEL
LIN {X 0,Y 145.511,Z 684.136,A -85,B 0,C 180,E1 -24186.586,E2 -24186.586} C_VEL
LIN {X 0,Y 142.395,Z 686.782,A -85,B 0,C 180,E1 -24192.773,E2 -24192.773} C_VEL
LIN {X 0,Y 141,Z 687.996,A -85,B 0,C 180,E1 -24198.498,E2 -24198.498} C_VEL
LIN {X 0,Y 140.76,Z 688.135,A -85,B 0,C 180,E1 -24204.268,E2 -24204.268} C_VEL
LIN {X 0,Y 140.97,Z 687.785,A -85,B 0,C 180,E1 -24207.141,E2 -24207.141} C_VEL
LIN {X 0,Y 141.188,Z 687.108,A -85,B 0,C 180,E1 -24209.999,E2 -24209.999} C_VEL
LIN {X 0,Y 140.957,Z 685.394,A -85,B 0,C 180,E1 -24214.315,E2 -24214.315} C_VEL
LIN {X 0,Y 140.969,Z 682.005,A -85,B 0,C 180,E1 -24220.048,E2 -24220.048} C_VEL
LIN {X 0,Y 141.999,Z 677.201,A -85,B 0,C 180,E1 -24225.795,E2 -24225.795} C_VEL
LIN {X 0,Y 144.187,Z 670.866,A -85,B 0,C 180,E1 -24231.441,E2 -24231.441} C_VEL
LIN {X 0,Y 147.058,Z 663.949,A -85,B 0,C 180,E1 -24236.234,E2 -24236.234} C_VEL
LIN {X 0,Y 150.91,Z 655.549,A -85,B 0,C 180,E1 -24240.814,E2 -24240.814} C_VEL
LIN {X 0,Y 155.476,Z 645.383,A -85,B 0,C 180,E1 -24245.192,E2 -24245.192} C_VEL
LIN {X 0,Y 160.232,Z 634.984,A -85,B 0,C 180,E1 -24248.682,E2 -24248.682} C_VEL
LIN {X 0,Y 165.516,Z 622.599,A -85,B 0,C 180,E1 -24251.97,E2 -24251.97} C_VEL
LIN {X 0,Y 170.365,Z 610.202,A -85,B 0,C 180,E1 -24254.529,E2 -24254.529} C_VEL
LIN {X 0,Y 174.459,Z 598.326,A -85,B 0,C 180,E1 -24256.477,E2 -24256.477} C_VEL
LIN {X 0,Y 178.789,Z 583.973,A -85,B 0,C 180,E1 -24258.318,E2 -24258.318} C_VEL
LIN {X 0,Y 182.5,Z 569.236,A -85,B 0,C 180,E1 -24259.725,E2 -24259.725} C_VEL
LIN {X 0,Y 185.199,Z 554.929,A -85,B 0,C 180,E1 -24260.748,E2 -24260.748} C_VEL
LIN {X 0,Y 187.169,Z 539.864,A -85,B 0,C 180,E1 -24261.503,E2 -24261.503} C_VEL
LIN {X 0,Y 193.43,Z 469.803,A -85,B 0,C 180,E1 -24263.996,E2 -24263.996} C_VEL
LIN {X 0,Y 187.102,Z 453.516,A -85,B 0,C 180,E1 -24266.889,E2 -24266.889} C_VEL
LIN {X 0,Y 180.658,Z 438.843,A -85,B 0,C 180,E1 -24270.026,E2 -24270.026} C_VEL
LIN {X 0,Y 174.963,Z 427.128,A -85,B 0,C 180,E1 -24273.055,E2 -24273.055} C_VEL
LIN {X 0,Y 169.892,Z 417.812,A -85,B 0,C 180,E1 -24275.92,E2 -24275.92} C_VEL
LIN {X 0,Y 165.515,Z 411.413,A -85,B 0,C 180,E1 -24278.558,E2 -24278.558} C_VEL
LIN {X 0,Y 162.322,Z 407.021,A -85,B 0,C 180,E1 -24280.611,E2 -24280.611} C_VEL
LIN {X 0,Y 159.266,Z 402.771,A -85,B 0,C 180,E1 -24282.755,E2 -24282.755} C_VEL
LIN {X 0,Y 156.589,Z 399.02,A -85,B 0,C 180,E1 -24284.796,E2 -24284.796} C_VEL
LIN {X 0,Y 153.573,Z 395.533,A -85,B 0,C 180,E1 -24287.232,E2 -24287.232} C_VEL
LIN {X 0,Y 152.467,Z 393.408,A -85,B 0,C 180,E1 -24288.291,E2 -24288.291} C_VEL
LIN {X 0,Y 149.864,Z 390.999,A -85,B 0,C 180,E1 -24290.632,E2 -24290.632} C_VEL
LIN {X 0,Y 148.321,Z 387.998,A -85,B 0,C 180,E1 -24292.343,E2 -24292.343} C_VEL
LIN {X 0,Y 145.633,Z 386.32,A -85,B 0,C 180,E1 -24295.156,E2 -24295.156} C_VEL
LIN {X 0,Y 144.263,Z 383.922,A -85,B 0,C 180,E1 -24297.034,E2 -24297.034} C_VEL
LIN {X 0,Y 143.889,Z 382.153,A -85,B 0,C 180,E1 -24297.902,E2 -24297.902} C_VEL
LIN {X 0,Y 144.175,Z 382.122,A -85,B 0,C 180,E1 -24300.001,E2 -24300.001} C_VEL
LIN {X 0,Y 143.681,Z 382.178,A -85,B 0,C 180,E1 -24308.439,E2 -24308.439} C_VEL
LIN {X 0,Y 143.57,Z 382.227,A -85,B 0,C 180,E1 -24311.759,E2 -24311.759} C_VEL
LIN {X 0,Y 143.302,Z 382.22,A -85,B 0,C 180,E1 -24317.114,E2 -24317.114} C_VEL
LIN {X 0,Y 143.274,Z 382.263,A -85,B 0,C 180,E1 -24321.254,E2 -24321.254} C_VEL
LIN {X 0,Y 143.189,Z 382.245,A -85,B 0,C 180,E1 -24327.938,E2 -24327.938} C_VEL
LIN {X 0,Y 143.146,Z 382.247,A -85,B 0,C 180,E1 -24333.424,E2 -24333.424} C_VEL
LIN {X 0,Y 143.056,Z 382.291,A -85,B 0,C 180,E1 -24339.693,E2 -24339.693} C_VEL
LIN {X 0,Y 143.054,Z 382.285,A -85,B 0,C 180,E1 -24342.441,E2 -24342.441} C_VEL
LIN {X 0,Y 143.597,Z 384.242,A -85,B 0,C 180,E1 -24343.425,E2 -24343.425} C_VEL
LIN {X 0,Y 145.453,Z 386.759,A -85,B 0,C 180,E1 -24345.886,E2 -24345.886} C_VEL
LIN {X 0,Y 147.952,Z 388.384,A -85,B 0,C 180,E1 -24348.528,E2 -24348.528} C_VEL
LIN {X 0,Y 149.291,Z 391.013,A -85,B 0,C 180,E1 -24350.044,E2 -24350.044} C_VEL
LIN {X 0,Y 151.974,Z 393.458,A -85,B 0,C 180,E1 -24352.505,E2 -24352.505} C_VEL
LIN {X 0,Y 152.498,Z 394.063,A -85,B 0,C 180,E1 -24352.975,E2 -24352.975} C_VEL
LIN {X 0,Y 154.829,Z 397.523,A -85,B 0,C 180,E1 -24355.03,E2 -24355.03} C_VEL
LIN {X 0,Y 156.631,Z 399.303,A -85,B 0,C 180,E1 -24356.4,E2 -24356.4} C_VEL
LIN {X 0,Y 159.406,Z 403.066,A -85,B 0,C 180,E1 -24358.502,E2 -24358.502} C_VEL
LIN {X 0,Y 163.956,Z 409.256,A -85,B 0,C 180,E1 -24361.608,E2 -24361.608} C_VEL
LIN {X 0,Y 169.599,Z 417.275,A -85,B 0,C 180,E1 -24365.037,E2 -24365.037} C_VEL
LIN {X 0,Y 176.761,Z 428.277,A -85,B 0,C 180,E1 -24368.877,E2 -24368.877} C_VEL
LIN {X 0,Y 182.813,Z 438.269,A -85,B 0,C 180,E1 -24371.814,E2 -24371.814} C_VEL
LIN {X 0,Y 191.921,Z 455.225,A -85,B 0,C 180,E1 -24375.804,E2 -24375.804} C_VEL
LIN {X 0,Y 193.561,Z 458.931,A -85,B 0,C 180,E1 -24376.503,E2 -24376.503} C_VEL
LIN {X 0,Y 187.457,Z 527.626,A -85,B 0,C 180,E1 -24379.001,E2 -24379.001} C_VEL
LIN {X 0,Y 185.244,Z 543.117,A -85,B 0,C 180,E1 -24379.917,E2 -24379.917} C_VEL
LIN {X 0,Y 182.173,Z 558.858,A -85,B 0,C 180,E1 -24381.264,E2 -24381.264} C_VEL
LIN {X 0,Y 178.484,Z 573.504,A -85,B 0,C 180,E1 -24382.933,E2 -24382.933} C_VEL
LIN {X 0,Y 174.471,Z 586.957,A -85,B 0,C 180,E1 -24384.921,E2 -24384.921} C_VEL
LIN {X 0,Y 169.914,Z 599.945,A -85,B 0,C 180,E1 -24387.334,E2 -24387.334} C_VEL
LIN {X 0,Y 164.948,Z 612.535,A -85,B 0,C 180,E1 -24390.306,E2 -24390.306} C_VEL
LIN {X 0,Y 159.985,Z 624.116,A -85,B 0,C 180,E1 -24393.779,E2 -24393.779} C_VEL
LIN {X 0,Y 155.153,Z 634.718,A -85,B 0,C 180,E1 -24397.811,E2 -24397.811} C_VEL
LIN {X 0,Y 150.936,Z 643.63,A -85,B 0,C 180,E1 -24402.085,E2 -24402.085} C_VEL
LIN {X 0,Y 147.097,Z 651.897,A -85,B 0,C 180,E1 -24407.141,E2 -24407.141} C_VEL
LIN {X 0,Y 144.266,Z 658.407,A -85,B 0,C 180,E1 -24412.238,E2 -24412.238} C_VEL
LIN {X 0,Y 142.362,Z 663.433,A -85,B 0,C 180,E1 -24417.298,E2 -24417.298} C_VEL
LIN {X 0,Y 140.886,Z 667.847,A -85,B 0,C 180,E1 -24423.281,E2 -24423.281} C_VEL
LIN {X 0,Y 140.504,Z 669.821,A -85,B 0,C 180,E1 -24426.889,E2 -24426.889} C_VEL
LIN {X 0,Y 140.507,Z 671.578,A -85,B 0,C 180,E1 -24431.383,E2 -24431.383} C_VEL
LIN {X 0,Y 141.036,Z 672.676,A -85,B 0,C 180,E1 -24435.761,E2 -24435.761} C_VEL
LIN {X 0,Y 142.634,Z 673.086,A -85,B 0,C 180,E1 -24442.035,E2 -24442.035} C_VEL
LIN {X 0,Y 145.398,Z 672.21,A -85,B 0,C 180,E1 -24447.878,E2 -24447.878} C_VEL
LIN {X 0,Y 149.285,Z 670.143,A -85,B 0,C 180,E1 -24453.443,E2 -24453.443} C_VEL
LIN {X 0,Y 154.22,Z 666.909,A -85,B 0,C 180,E1 -24458.618,E2 -24458.618} C_VEL
LIN {X 0,Y 159.673,Z 662.895,A -85,B 0,C 180,E1 -24463.015,E2 -24463.015} C_VEL
LIN {X 0,Y 167.292,Z 656.589,A -85,B 0,C 180,E1 -24467.874,E2 -24467.874} C_VEL
LIN {X 0,Y 175.011,Z 649.46,A -85,B 0,C 180,E1 -24471.823,E2 -24471.823} C_VEL
LIN {X 0,Y 183.841,Z 640.185,A -85,B 0,C 180,E1 -24475.614,E2 -24475.614} C_VEL
LIN {X 0,Y 191.654,Z 631.074,A -85,B 0,C 180,E1 -24478.423,E2 -24478.423} C_VEL
LIN {X 0,Y 199.19,Z 621.138,A -85,B 0,C 180,E1 -24480.82,E2 -24480.82} C_VEL
LIN {X 0,Y 207.037,Z 609.292,A -85,B 0,C 180,E1 -24483.017,E2 -24483.017} C_VEL
LIN {X 0,Y 214.602,Z 595.971,A -85,B 0,C 180,E1 -24484.944,E2 -24484.944} C_VEL
LIN {X 0,Y 220.73,Z 583.263,A -85,B 0,C 180,E1 -24486.381,E2 -24486.381} C_VEL
LIN {X 0,Y 226.159,Z 569.703,A -85,B 0,C 180,E1 -24487.573,E2 -24487.573} C_VEL
LIN {X 0,Y 230.827,Z 554.92,A -85,B 0,C 180,E1 -24488.603,E2 -24488.603} C_VEL
LIN {X 0,Y 234.478,Z 539.627,A -85,B 0,C 180,E1 -24489.357,E2 -24489.357} C_VEL
LIN {X 0,Y 237.206,Z 522.876,A -85,B 0,C 180,E1 -24489.9,E2 -24489.9} C_VEL
LIN {X 0,Y 241.637,Z 488.691,A -85,B 0,C 180,E1 -24490.87,E2 -24490.87} C_VEL
LIN {X 0,Y 240.558,Z 486.085,A -85,B 0,C 180,E1 -24492.671,E2 -24492.671} C_VEL
LIN {X 0,Y 239.81,Z 484.04,A -85,B 0,C 180,E1 -24494.428,E2 -24494.428} C_VEL
LIN {X 0,Y 238.889,Z 481.291,A -85,B 0,C 180,E1 -24498.881,E2 -24498.881} C_VEL
LIN {X 0,Y 238.914,Z 482.503,A -85,B 0,C 180,E1 -24501.648,E2 -24501.648} C_VEL
LIN {X 0,Y 239.631,Z 486.475,A -85,B 0,C 180,E1 -24505.068,E2 -24505.068} C_VEL
LIN {X 0,Y 240.449,Z 490.354,A -85,B 0,C 180,E1 -24507.157,E2 -24507.157} C_VEL
LIN {X 0,Y 241.151,Z 493.699,A -85,B 0,C 180,E1 -24508.584,E2 -24508.584} C_VEL
LIN {X 0,Y 234.964,Z 539.729,A -85,B 0,C 180,E1 -24509.839,E2 -24509.839} C_VEL
LIN {X 0,Y 231.557,Z 555.626,A -85,B 0,C 180,E1 -24510.439,E2 -24510.439} C_VEL
LIN {X 0,Y 227.268,Z 570.038,A -85,B 0,C 180,E1 -24511.106,E2 -24511.106} C_VEL
LIN {X 0,Y 222.521,Z 582.844,A -85,B 0,C 180,E1 -24511.917,E2 -24511.917} C_VEL
LIN {X 0,Y 216.082,Z 597.225,A -85,B 0,C 180,E1 -24513.12,E2 -24513.12} C_VEL
LIN {X 0,Y 209.083,Z 610.323,A -85,B 0,C 180,E1 -24514.559,E2 -24514.559} C_VEL
LIN {X 0,Y 201.033,Z 623.474,A -85,B 0,C 180,E1 -24516.478,E2 -24516.478} C_VEL
LIN {X 0,Y 191.983,Z 636.214,A -85,B 0,C 180,E1 -24518.929,E2 -24518.929} C_VEL
LIN {X 0,Y 183.491,Z 646.821,A -85,B 0,C 180,E1 -24521.678,E2 -24521.678} C_VEL
LIN {X 0,Y 176.762,Z 654.506,A -85,B 0,C 180,E1 -24524.262,E2 -24524.262} C_VEL
LIN {X 0,Y 173.268,Z 657.845,A -85,B 0,C 180,E1 -24525.379,E2 -24525.379} C_VEL
LIN {X 0,Y 166.276,Z 663.045,A -85,B 0,C 180,E1 -24526.979,E2 -24526.979} C_VEL
LIN {X 0,Y 159.296,Z 667.789,A -85,B 0,C 180,E1 -24528.802,E2 -24528.802} C_VEL
LIN {X 0,Y 155.894,Z 670.318,A -85,B 0,C 180,E1 -24530.273,E2 -24530.273} C_VEL
LIN {X 0,Y 148.467,Z 676.552,A -85,B 0,C 180,E1 -24535.385,E2 -24535.385} C_VEL
LIN {X 0,Y 142.856,Z 681.002,A -85,B 0,C 180,E1 -24540.529,E2 -24540.529} C_VEL
LIN {X 0,Y 138.534,Z 684.321,A -85,B 0,C 180,E1 -24546.054,E2 -24546.054} C_VEL
LIN {X 0,Y 135.564,Z 686.52,A -85,B 0,C 180,E1 -24551.876,E2 -24551.876} C_VEL
LIN {X 0,Y 133.989,Z 687.606,A -85,B 0,C 180,E1 -24557.887,E2 -24557.887} C_VEL
LIN {X 0,Y 133.676,Z 687.622,A -85,B 0,C 180,E1 -24563.963,E2 -24563.963} C_VEL
LIN {X 0,Y 133.892,Z 687.214,A -85,B 0,C 180,E1 -24566.99,E2 -24566.99} C_VEL
LIN {X 0,Y 134.125,Z 686.503,A -85,B 0,C 180,E1 -24569.999,E2 -24569.999} C_VEL
LIN {X 0,Y 133.891,Z 684.868,A -85,B 0,C 180,E1 -24574.211,E2 -24574.211} C_VEL
LIN {X 0,Y 133.957,Z 681.201,A -85,B 0,C 180,E1 -24580.58,E2 -24580.58} C_VEL
LIN {X 0,Y 135.129,Z 676.263,A -85,B 0,C 180,E1 -24586.62,E2 -24586.62} C_VEL
LIN {X 0,Y 137.456,Z 669.93,A -85,B 0,C 180,E1 -24592.419,E2 -24592.419} C_VEL
LIN {X 0,Y 140.629,Z 662.719,A -85,B 0,C 180,E1 -24597.532,E2 -24597.532} C_VEL
LIN {X 0,Y 144.761,Z 654.17,A -85,B 0,C 180,E1 -24602.277,E2 -24602.277} C_VEL
LIN {X 0,Y 149.425,Z 644.264,A -85,B 0,C 180,E1 -24606.6,E2 -24606.6} C_VEL
LIN {X 0,Y 154.65,Z 633.178,A -85,B 0,C 180,E1 -24610.358,E2 -24610.358} C_VEL
LIN {X 0,Y 159.758,Z 621.663,A -85,B 0,C 180,E1 -24613.421,E2 -24613.421} C_VEL
LIN {X 0,Y 164.798,Z 609.175,A -85,B 0,C 180,E1 -24616.024,E2 -24616.024} C_VEL
LIN {X 0,Y 169.589,Z 595.572,A -85,B 0,C 180,E1 -24618.238,E2 -24618.238} C_VEL
LIN {X 0,Y 174.07,Z 580.554,A -85,B 0,C 180,E1 -24620.094,E2 -24620.094} C_VEL
LIN {X 0,Y 177.765,Z 565.558,A -85,B 0,C 180,E1 -24621.448,E2 -24621.448} C_VEL
LIN {X 0,Y 180.591,Z 550.046,A -85,B 0,C 180,E1 -24622.458,E2 -24622.458} C_VEL
LIN {X 0,Y 182.442,Z 533.951,A -85,B 0,C 180,E1 -24623.179,E2 -24623.179} C_VEL
LIN {X 0,Y 188.075,Z 471.832,A -85,B 0,C 180,E1 -24625.418,E2 -24625.418} C_VEL
LIN {X 0,Y 182.614,Z 457.449,A -85,B 0,C 180,E1 -24628.081,E2 -24628.081} C_VEL
LIN {X 0,Y 176.587,Z 443.347,A -85,B 0,C 180,E1 -24631.194,E2 -24631.194} C_VEL
LIN {X 0,Y 171.237,Z 432.128,A -85,B 0,C 180,E1 -24634.176,E2 -24634.176} C_VEL
LIN {X 0,Y 166.451,Z 423.045,A -85,B 0,C 180,E1 -24637.069,E2 -24637.069} C_VEL
LIN {X 0,Y 162.1,Z 416.658,A -85,B 0,C 180,E1 -24639.816,E2 -24639.816} C_VEL
LIN {X 0,Y 159.222,Z 412.581,A -85,B 0,C 180,E1 -24641.78,E2 -24641.78} C_VEL
LIN {X 0,Y 156.544,Z 408.69,A -85,B 0,C 180,E1 -24643.786,E2 -24643.786} C_VEL
LIN {X 0,Y 153.478,Z 404.55,A -85,B 0,C 180,E1 -24646.238,E2 -24646.238} C_VEL
LIN {X 0,Y 150.872,Z 401.197,A -85,B 0,C 180,E1 -24648.506,E2 -24648.506} C_VEL
LIN {X 0,Y 149.828,Z 399.557,A -85,B 0,C 180,E1 -24649.529,E2 -24649.529} C_VEL
LIN {X 0,Y 147.2,Z 396.551,A -85,B 0,C 180,E1 -24652.111,E2 -24652.111} C_VEL
LIN {X 0,Y 146.224,Z 394.649,A -85,B 0,C 180,E1 -24653.273,E2 -24653.273} C_VEL
LIN {X 0,Y 143.668,Z 392.696,A -85,B 0,C 180,E1 -24656.144,E2 -24656.144} C_VEL
LIN {X 0,Y 142.201,Z 389.929,A -85,B 0,C 180,E1 -24658.319,E2 -24658.319} C_VEL
LIN {X 0,Y 141.843,Z 388.896,A -85,B 0,C 180,E1 -24658.936,E2 -24658.936} C_VEL
LIN {X 0,Y 138.029,Z 386.54,A -85,B 0,C 180,E1 -24665.113,E2 -24665.113} C_VEL
LIN {X 0,Y 136.849,Z 384.2,A -85,B 0,C 180,E1 -24668.12,E2 -24668.12} C_VEL
LIN {X 0,Y 136.582,Z 383.068,A -85,B 0,C 180,E1 -24669.254,E2 -24669.254} C_VEL
LIN {X 0,Y 136.49,Z 383.109,A -85,B 0,C 180,E1 -24671.958,E2 -24671.958} C_VEL
LIN {X 0,Y 136.242,Z 383.104,A -85,B 0,C 180,E1 -24678.031,E2 -24678.031} C_VEL
LIN {X 0,Y 136.195,Z 383.142,A -85,B 0,C 180,E1 -24681.748,E2 -24681.748} C_VEL
LIN {X 0,Y 136.1,Z 383.135,A -85,B 0,C 180,E1 -24688.619,E2 -24688.619} C_VEL
LIN {X 0,Y 136.078,Z 383.336,A -85,B 0,C 180,E1 -24690.749,E2 -24690.749} C_VEL
LIN {X 0,Y 137.646,Z 386.791,A -85,B 0,C 180,E1 -24695.462,E2 -24695.462} C_VEL
LIN {X 0,Y 140.096,Z 388.74,A -85,B 0,C 180,E1 -24699.918,E2 -24699.918} C_VEL
LIN {X 0,Y 141.207,Z 389.26,A -85,B 0,C 180,E1 -24701.516,E2 -24701.516} C_VEL
LIN {X 0,Y 142.475,Z 391.925,A -85,B 0,C 180,E1 -24703.534,E2 -24703.534} C_VEL
LIN {X 0,Y 144.981,Z 394.387,A -85,B 0,C 180,E1 -24706.648,E2 -24706.648} C_VEL
LIN {X 0,Y 145.92,Z 395.091,A -85,B 0,C 180,E1 -24707.665,E2 -24707.665} C_VEL
LIN {X 0,Y 147.88,Z 398.249,A -85,B 0,C 180,E1 -24709.858,E2 -24709.858} C_VEL
LIN {X 0,Y 150.261,Z 400.487,A -85,B 0,C 180,E1 -24712.085,E2 -24712.085} C_VEL
LIN {X 0,Y 152.616,Z 403.943,A -85,B 0,C 180,E1 -24714.26,E2 -24714.26} C_VEL
LIN {X 0,Y 154.198,Z 405.637,A -85,B 0,C 180,E1 -24715.532,E2 -24715.532} C_VEL
LIN {X 0,Y 157.936,Z 410.832,A -85,B 0,C 180,E1 -24718.429,E2 -24718.429} C_VEL
LIN {X 0,Y 161.164,Z 415.315,A -85,B 0,C 180,E1 -24720.712,E2 -24720.712} C_VEL
LIN {X 0,Y 166.641,Z 423.267,A -85,B 0,C 180,E1 -24724.174,E2 -24724.174} C_VEL
LIN {X 0,Y 173.357,Z 433.849,A -85,B 0,C 180,E1 -24727.966,E2 -24727.966} C_VEL
LIN {X 0,Y 179.028,Z 443.432,A -85,B 0,C 180,E1 -24730.842,E2 -24730.842} C_VEL
LIN {X 0,Y 187.652,Z 459.869,A -85,B 0,C 180,E1 -24734.802,E2 -24734.802} C_VEL
LIN {X 0,Y 188.297,Z 461.371,A -85,B 0,C 180,E1 -24735.098,E2 -24735.098} C_VEL
LIN {X 0,Y 182.171,Z 527.85,A -85,B 0,C 180,E1 -24737.538,E2 -24737.538} C_VEL
LIN {X 0,Y 179.792,Z 543.741,A -85,B 0,C 180,E1 -24738.483,E2 -24738.483} C_VEL
LIN {X 0,Y 176.899,Z 558.366,A -85,B 0,C 180,E1 -24739.746,E2 -24739.746} C_VEL
LIN {X 0,Y 173.173,Z 572.885,A -85,B 0,C 180,E1 -24741.394,E2 -24741.394} C_VEL
LIN {X 0,Y 168.926,Z 586.68,A -85,B 0,C 180,E1 -24743.43,E2 -24743.43} C_VEL
LIN {X 0,Y 163.993,Z 600.32,A -85,B 0,C 180,E1 -24746.008,E2 -24746.008} C_VEL
LIN {X 0,Y 158.823,Z 612.924,A -85,B 0,C 180,E1 -24749.05,E2 -24749.05} C_VEL
LIN {X 0,Y 153.639,Z 624.512,A -85,B 0,C 180,E1 -24752.623,E2 -24752.623} C_VEL
LIN {X 0,Y 148.625,Z 635.05,A -85,B 0,C 180,E1 -24756.763,E2 -24756.763} C_VEL
LIN {X 0,Y 144.182,Z 644.044,A -85,B 0,C 180,E1 -24761.245,E2 -24761.245} C_VEL
LIN {X 0,Y 140.699,Z 651.254,A -85,B 0,C 180,E1 -24765.752,E2 -24765.752} C_VEL
LIN {X 0,Y 137.674,Z 657.796,A -85,B 0,C 180,E1 -24770.938,E2 -24770.938} C_VEL
LIN {X 0,Y 135.591,Z 662.861,A -85,B 0,C 180,E1 -24776.077,E2 -24776.077} C_VEL
LIN {X 0,Y 134.087,Z 667.072,A -85,B 0,C 180,E1 -24781.612,E2 -24781.612} C_VEL
LIN {X 0,Y 133.344,Z 670.431,A -85,B 0,C 180,E1 -24787.758,E2 -24787.758} C_VEL
LIN {X 0,Y 133.552,Z 672.352,A -85,B 0,C 180,E1 -24793.167,E2 -24793.167} C_VEL
LIN {X 0,Y 134.173,Z 673.213,A -85,B 0,C 180,E1 -24797.167,E2 -24797.167} C_VEL
LIN {X 0,Y 135.277,Z 673.546,A -85,B 0,C 180,E1 -24801.431,E2 -24801.431} C_VEL
LIN {X 0,Y 136.983,Z 673.332,A -85,B 0,C 180,E1 -24805.641,E2 -24805.641} C_VEL
LIN {X 0,Y 139.219,Z 672.599,A -85,B 0,C 180,E1 -24809.679,E2 -24809.679} C_VEL
LIN {X 0,Y 141.966,Z 671.354,A -85,B 0,C 180,E1 -24813.541,E2 -24813.541} C_VEL
LIN {X 0,Y 147.058,Z 668.43,A -85,B 0,C 180,E1 -24818.997,E2 -24818.997} C_VEL
LIN {X 0,Y 153.417,Z 664.188,A -85,B 0,C 180,E1 -24824.16,E2 -24824.16} C_VEL
LIN {X 0,Y 160.739,Z 658.67,A -85,B 0,C 180,E1 -24828.776,E2 -24828.776} C_VEL
LIN {X 0,Y 168.661,Z 651.951,A -85,B 0,C 180,E1 -24832.818,E2 -24832.818} C_VEL
LIN {X 0,Y 176.712,Z 644.307,A -85,B 0,C 180,E1 -24836.27,E2 -24836.27} C_VEL
LIN {X 0,Y 184.927,Z 635.54,A -85,B 0,C 180,E1 -24839.271,E2 -24839.271} C_VEL
LIN {X 0,Y 193.959,Z 624.598,A -85,B 0,C 180,E1 -24842.076,E2 -24842.076} C_VEL
LIN {X 0,Y 202.149,Z 613.245,A -85,B 0,C 180,E1 -24844.301,E2 -24844.301} C_VEL
LIN {X 0,Y 209.561,Z 601.321,A -85,B 0,C 180,E1 -24846.121,E2 -24846.121} C_VEL
LIN {X 0,Y 216.223,Z 588.697,A -85,B 0,C 180,E1 -24847.659,E2 -24847.659} C_VEL
LIN {X 0,Y 222.209,Z 575.228,A -85,B 0,C 180,E1 -24848.919,E2 -24848.919} C_VEL
LIN {X 0,Y 227.447,Z 560.637,A -85,B 0,C 180,E1 -24849.996,E2 -24849.996} C_VEL
LIN {X 0,Y 231.541,Z 545.897,A -85,B 0,C 180,E1 -24850.792,E2 -24850.792} C_VEL
LIN {X 0,Y 234.467,Z 531.309,A -85,B 0,C 180,E1 -24851.352,E2 -24851.352} C_VEL
LIN {X 0,Y 239.588,Z 493.633,A -85,B 0,C 180,E1 -24852.409,E2 -24852.409} C_VEL
LIN {X 0,Y 238.499,Z 490.791,A -85,B 0,C 180,E1 -24854.97,E2 -24854.97} C_VEL
LIN {X 0,Y 237.803,Z 488.357,A -85,B 0,C 180,E1 -24858.971,E2 -24858.971} C_VEL
LIN {X 0,Y 237.8,Z 489.459,A -85,B 0,C 180,E1 -24861.37,E2 -24861.37} C_VEL
LIN {X 0,Y 238.343,Z 493.175,A -85,B 0,C 180,E1 -24864.576,E2 -24864.576} C_VEL
LIN {X 0,Y 238.949,Z 496.711,A -85,B 0,C 180,E1 -24866.489,E2 -24866.489} C_VEL
LIN {X 0,Y 239.159,Z 498.213,A -85,B 0,C 180,E1 -24867.065,E2 -24867.065} C_VEL
LIN {X 0,Y 233.465,Z 539.104,A -85,B 0,C 180,E1 -24868.134,E2 -24868.134} C_VEL
LIN {X 0,Y 230.246,Z 553.885,A -85,B 0,C 180,E1 -24868.649,E2 -24868.649} C_VEL
LIN {X 0,Y 225.713,Z 568.971,A -85,B 0,C 180,E1 -24869.326,E2 -24869.326} C_VEL
LIN {X 0,Y 220.448,Z 582.73,A -85,B 0,C 180,E1 -24870.143,E2 -24870.143} C_VEL
LIN {X 0,Y 213.857,Z 597.049,A -85,B 0,C 180,E1 -24871.301,E2 -24871.301} C_VEL
LIN {X 0,Y 207.349,Z 608.89,A -85,B 0,C 180,E1 -24872.527,E2 -24872.527} C_VEL
LIN {X 0,Y 199.433,Z 621.502,A -85,B 0,C 180,E1 -24874.271,E2 -24874.271} C_VEL
LIN {X 0,Y 191.627,Z 632.354,A -85,B 0,C 180,E1 -24876.208,E2 -24876.208} C_VEL
LIN {X 0,Y 183.9,Z 642.042,A -85,B 0,C 180,E1 -24878.422,E2 -24878.422} C_VEL
LIN {X 0,Y 177.698,Z 649.071,A -85,B 0,C 180,E1 -24880.416,E2 -24880.416} C_VEL
LIN {X 0,Y 169.547,Z 657.588,A -85,B 0,C 180,E1 -24883.496,E2 -24883.496} C_VEL
LIN {X 0,Y 160.983,Z 665.743,A -85,B 0,C 180,E1 -24887.414,E2 -24887.414} C_VEL
LIN {X 0,Y 155.894,Z 670.318,A -85,B 0,C 180,E1 -24890.273,E2 -24890.273} C_VEL
LIN {X 0,Y 152.551,Z 672.749,A -85,B 0,C 180,E1 -24891.848,E2 -24891.848} C_VEL
LIN {X 0,Y 143.125,Z 677.702,A -85,B 0,C 180,E1 -24895.311,E2 -24895.311} C_VEL
LIN {X 0,Y 138.341,Z 680.022,A -85,B 0,C 180,E1 -24897.688,E2 -24897.688} C_VEL
LIN {X 0,Y 136.602,Z 681.012,A -85,B 0,C 180,E1 -24899.099,E2 -24899.099} C_VEL
LIN {X 0,Y 131.875,Z 684.21,A -85,B 0,C 180,E1 -24904.953,E2 -24904.953} C_VEL
LIN {X 0,Y 128.776,Z 686.234,A -85,B 0,C 180,E1 -24910.884,E2 -24910.884} C_VEL
LIN {X 0,Y 126.978,Z 687.217,A -85,B 0,C 180,E1 -24917.208,E2 -24917.208} C_VEL
LIN {X 0,Y 126.594,Z 687.108,A -85,B 0,C 180,E1 -24923.624,E2 -24923.624} C_VEL
LIN {X 0,Y 126.826,Z 686.641,A -85,B 0,C 180,E1 -24926.822,E2 -24926.822} C_VEL
LIN {X 0,Y 127.061,Z 685.867,A -85,B 0,C 180,E1 -24929.999,E2 -24929.999} C_VEL
LIN {X 0,Y 126.816,Z 684.347,A -85,B 0,C 180,E1 -24934.037,E2 -24934.037} C_VEL
LIN {X 0,Y 126.786,Z 681.432,A -85,B 0,C 180,E1 -24939.571,E2 -24939.571} C_VEL
LIN {X 0,Y 127.782,Z 676.722,A -85,B 0,C 180,E1 -24945.961,E2 -24945.961} C_VEL
LIN {X 0,Y 130.11,Z 670.494,A -85,B 0,C 180,E1 -24952.215,E2 -24952.215} C_VEL
LIN {X 0,Y 133.21,Z 663.646,A -85,B 0,C 180,E1 -24957.491,E2 -24957.491} C_VEL
LIN {X 0,Y 137.36,Z 655.36,A -85,B 0,C 180,E1 -24962.494,E2 -24962.494} C_VEL
LIN {X 0,Y 142.213,Z 645.542,A -85,B 0,C 180,E1 -24967.131,E2 -24967.131} C_VEL
LIN {X 0,Y 147.422,Z 635.078,A -85,B 0,C 180,E1 -24970.956,E2 -24970.956} C_VEL
LIN {X 0,Y 153.085,Z 622.873,A -85,B 0,C 180,E1 -24974.434,E2 -24974.434} C_VEL
LIN {X 0,Y 158.265,Z 610.702,A -85,B 0,C 180,E1 -24977.112,E2 -24977.112} C_VEL
LIN {X 0,Y 162.645,Z 599.127,A -85,B 0,C 180,E1 -24979.128,E2 -24979.128} C_VEL
LIN {X 0,Y 167.416,Z 584.466,A -85,B 0,C 180,E1 -24981.118,E2 -24981.118} C_VEL
LIN {X 0,Y 171.407,Z 569.726,A -85,B 0,C 180,E1 -24982.598,E2 -24982.598} C_VEL
LIN {X 0,Y 174.43,Z 555.072,A -85,B 0,C 180,E1 -24983.688,E2 -24983.688} C_VEL
LIN {X 0,Y 176.676,Z 539.233,A -85,B 0,C 180,E1 -24984.509,E2 -24984.509} C_VEL
LIN {X 0,Y 182.937,Z 474.051,A -85,B 0,C 180,E1 -24986.878,E2 -24986.878} C_VEL
LIN {X 0,Y 177.263,Z 459.123,A -85,B 0,C 180,E1 -24989.8,E2 -24989.8} C_VEL
LIN {X 0,Y 171.026,Z 444.455,A -85,B 0,C 180,E1 -24993.292,E2 -24993.292} C_VEL
LIN {X 0,Y 165.427,Z 432.708,A -85,B 0,C 180,E1 -24996.713,E2 -24996.713} C_VEL
LIN {X 0,Y 162.321,Z 427.031,A -85,B 0,C 180,E1 -24998.742,E2 -24998.742} C_VEL
LIN {X 0,Y 156.305,Z 418.264,A -85,B 0,C 180,E1 -25002.913,E2 -25002.913} C_VEL
LIN {X 0,Y 153.499,Z 414.207,A -85,B 0,C 180,E1 -25005.127,E2 -25005.127} C_VEL
LIN {X 0,Y 151.08,Z 410.8,A -85,B 0,C 180,E1 -25007.164,E2 -25007.164} C_VEL
LIN {X 0,Y 148.357,Z 407.021,A -85,B 0,C 180,E1 -25009.715,E2 -25009.715} C_VEL
LIN {X 0,Y 147.518,Z 405.841,A -85,B 0,C 180,E1 -25010.561,E2 -25010.561} C_VEL
LIN {X 0,Y 144.833,Z 402.389,A -85,B 0,C 180,E1 -25013.405,E2 -25013.405} C_VEL
LIN {X 0,Y 144.315,Z 401.335,A -85,B 0,C 180,E1 -25014.061,E2 -25014.061} C_VEL
LIN {X 0,Y 141.827,Z 399.171,A -85,B 0,C 180,E1 -25017.05,E2 -25017.05} C_VEL
LIN {X 0,Y 140.218,Z 396.055,A -85,B 0,C 180,E1 -25019.552,E2 -25019.552} C_VEL
LIN {X 0,Y 139.946,Z 395.563,A -85,B 0,C 180,E1 -25020.001,E2 -25020.001} C_VEL
LIN {X 0,Y 136.644,Z 393.349,A -85,B 0,C 180,E1 -25025.72,E2 -25025.72} C_VEL
LIN {X 0,Y 135.437,Z 390.777,A -85,B 0,C 180,E1 -25029.088,E2 -25029.088} C_VEL
LIN {X 0,Y 135.274,Z 390.057,A -85,B 0,C 180,E1 -25029.789,E2 -25029.789} C_VEL
LIN {X 0,Y 133.371,Z 389.653,A -85,B 0,C 180,E1 -25041.647,E2 -25041.647} C_VEL
LIN {X 0,Y 134.822,Z 390.241,A -85,B 0,C 180,E1 -25050.116,E2 -25050.116} C_VEL
LIN {X 0,Y 136.337,Z 393.682,A -85,B 0,C 180,E1 -25054.995,E2 -25054.995} C_VEL
LIN {X 0,Y 138.78,Z 395.671,A -85,B 0,C 180,E1 -25059.584,E2 -25059.584} C_VEL
LIN {X 0,Y 139.565,Z 396.198,A -85,B 0,C 180,E1 -25060.794,E2 -25060.794} C_VEL
LIN {X 0,Y 141.065,Z 398.97,A -85,B 0,C 180,E1 -25063.2,E2 -25063.2} C_VEL
LIN {X 0,Y 144.043,Z 401.887,A -85,B 0,C 180,E1 -25066.917,E2 -25066.917} C_VEL
LIN {X 0,Y 146.351,Z 405.246,A -85,B 0,C 180,E1 -25069.537,E2 -25069.537} C_VEL
LIN {X 0,Y 148.159,Z 407.06,A -85,B 0,C 180,E1 -25071.271,E2 -25071.271} C_VEL
LIN {X 0,Y 150.759,Z 410.715,A -85,B 0,C 180,E1 -25073.75,E2 -25073.75} C_VEL
LIN {X 0,Y 152.133,Z 412.46,A -85,B 0,C 180,E1 -25074.928,E2 -25074.928} C_VEL
LIN {X 0,Y 155.423,Z 417.072,A -85,B 0,C 180,E1 -25077.554,E2 -25077.554} C_VEL
LIN {X 0,Y 160.159,Z 423.794,A -85,B 0,C 180,E1 -25080.987,E2 -25080.987} C_VEL
LIN {X 0,Y 166.644,Z 433.954,A -85,B 0,C 180,E1 -25085.098,E2 -25085.098} C_VEL
LIN {X 0,Y 174.046,Z 446.234,A -85,B 0,C 180,E1 -25089.173,E2 -25089.173} C_VEL
LIN {X 0,Y 183.057,Z 463.669,A -85,B 0,C 180,E1 -25093.606,E2 -25093.606} C_VEL
LIN {X 0,Y 176.887,Z 528.655,A -85,B 0,C 180,E1 -25096.045,E2 -25096.045} C_VEL
LIN {X 0,Y 174.396,Z 544.394,A -85,B 0,C 180,E1 -25096.988,E2 -25096.988} C_VEL
LIN {X 0,Y 171.334,Z 559.339,A -85,B 0,C 180,E1 -25098.316,E2 -25098.316} C_VEL
LIN {X 0,Y 167.357,Z 574.058,A -85,B 0,C 180,E1 -25100.026,E2 -25100.026} C_VEL
LIN {X 0,Y 162.883,Z 588.01,A -85,B 0,C 180,E1 -25102.161,E2 -25102.161} C_VEL
LIN {X 0,Y 158.152,Z 600.554,A -85,B 0,C 180,E1 -25104.583,E2 -25104.583} C_VEL
LIN {X 0,Y 152.777,Z 613.176,A -85,B 0,C 180,E1 -25107.694,E2 -25107.694} C_VEL
LIN {X 0,Y 147.623,Z 624.317,A -85,B 0,C 180,E1 -25111.198,E2 -25111.198} C_VEL
LIN {X 0,Y 142.086,Z 635.424,A -85,B 0,C 180,E1 -25115.679,E2 -25115.679} C_VEL
LIN {X 0,Y 137.611,Z 644.154,A -85,B 0,C 180,E1 -25120.179,E2 -25120.179} C_VEL
LIN {X 0,Y 133.666,Z 651.905,A -85,B 0,C 180,E1 -25125.243,E2 -25125.243} C_VEL
LIN {X 0,Y 130.657,Z 658.163,A -85,B 0,C 180,E1 -25130.466,E2 -25130.466} C_VEL
LIN {X 0,Y 128.458,Z 663.31,A -85,B 0,C 180,E1 -25135.958,E2 -25135.958} C_VEL
LIN {X 0,Y 126.953,Z 667.455,A -85,B 0,C 180,E1 -25141.696,E2 -25141.696} C_VEL
LIN {X 0,Y 126.224,Z 671.063,A -85,B 0,C 180,E1 -25148.783,E2 -25148.783} C_VEL
LIN {X 0,Y 126.503,Z 672.719,A -85,B 0,C 180,E1 -25153.76,E2 -25153.76} C_VEL
LIN {X 0,Y 127.785,Z 673.859,A -85,B 0,C 180,E1 -25160.354,E2 -25160.354} C_VEL
LIN {X 0,Y 130.645,Z 673.751,A -85,B 0,C 180,E1 -25167.455,E2 -25167.455} C_VEL
LIN {X 0,Y 134.13,Z 672.611,A -85,B 0,C 180,E1 -25172.97,E2 -25172.97} C_VEL
LIN {X 0,Y 137.462,Z 671.094,A -85,B 0,C 180,E1 -25176.97,E2 -25176.97} C_VEL
LIN {X 0,Y 143.996,Z 667.488,A -85,B 0,C 180,E1 -25182.971,E2 -25182.971} C_VEL
LIN {X 0,Y 150.964,Z 662.963,A -85,B 0,C 180,E1 -25187.865,E2 -25187.865} C_VEL
LIN {X 0,Y 159.181,Z 656.954,A -85,B 0,C 180,E1 -25192.388,E2 -25192.388} C_VEL
LIN {X 0,Y 167.363,Z 650.213,A -85,B 0,C 180,E1 -25196.045,E2 -25196.045} C_VEL
LIN {X 0,Y 175.716,Z 642.365,A -85,B 0,C 180,E1 -25199.292,E2 -25199.292} C_VEL
LIN {X 0,Y 184.649,Z 632.981,A -85,B 0,C 180,E1 -25202.181,E2 -25202.181} C_VEL
LIN {X 0,Y 193.474,Z 622.348,A -85,B 0,C 180,E1 -25204.664,E2 -25204.664} C_VEL
LIN {X 0,Y 201.849,Z 610.664,A -85,B 0,C 180,E1 -25206.749,E2 -25206.749} C_VEL
LIN {X 0,Y 210.258,Z 596.873,A -85,B 0,C 180,E1 -25208.651,E2 -25208.651} C_VEL
LIN {X 0,Y 217.005,Z 583.731,A -85,B 0,C 180,E1 -25210.024,E2 -25210.024} C_VEL
LIN {X 0,Y 223.019,Z 569.416,A -85,B 0,C 180,E1 -25211.178,E2 -25211.178} C_VEL
LIN {X 0,Y 227.467,Z 556.169,A -85,B 0,C 180,E1 -25212.037,E2 -25212.037} C_VEL
LIN {X 0,Y 231.395,Z 540.795,A -85,B 0,C 180,E1 -25212.75,E2 -25212.75} C_VEL
LIN {X 0,Y 234.264,Z 524.315,A -85,B 0,C 180,E1 -25213.254,E2 -25213.254} C_VEL
LIN {X 0,Y 237.747,Z 499.071,A -85,B 0,C 180,E1 -25213.96,E2 -25213.96} C_VEL
LIN {X 0,Y 237.303,Z 497.709,A -85,B 0,C 180,E1 -25215.253,E2 -25215.253} C_VEL
LIN {X 0,Y 236.711,Z 495.436,A -85,B 0,C 180,E1 -25219.061,E2 -25219.061} C_VEL
LIN {X 0,Y 236.694,Z 496.411,A -85,B 0,C 180,E1 -25221.109,E2 -25221.109} C_VEL
LIN {X 0,Y 237.054,Z 499.758,A -85,B 0,C 180,E1 -25224,E2 -25224} C_VEL
LIN {X 0,Y 237.407,Z 502.433,A -85,B 0,C 180,E1 -25225.484,E2 -25225.484} C_VEL
LIN {X 0,Y 232.002,Z 539.483,A -85,B 0,C 180,E1 -25226.428,E2 -25226.428} C_VEL
LIN {X 0,Y 228.609,Z 554.4,A -85,B 0,C 180,E1 -25226.932,E2 -25226.932} C_VEL
LIN {X 0,Y 224.36,Z 568.218,A -85,B 0,C 180,E1 -25227.515,E2 -25227.515} C_VEL
LIN {X 0,Y 218.61,Z 582.921,A -85,B 0,C 180,E1 -25228.348,E2 -25228.348} C_VEL
LIN {X 0,Y 211.857,Z 597.016,A -85,B 0,C 180,E1 -25229.447,E2 -25229.447} C_VEL
LIN {X 0,Y 204.448,Z 609.945,A -85,B 0,C 180,E1 -25230.751,E2 -25230.751} C_VEL
LIN {X 0,Y 195.898,Z 622.911,A -85,B 0,C 180,E1 -25232.534,E2 -25232.534} C_VEL
LIN {X 0,Y 187.591,Z 633.827,A -85,B 0,C 180,E1 -25234.489,E2 -25234.489} C_VEL
LIN {X 0,Y 180.91,Z 641.698,A -85,B 0,C 180,E1 -25236.282,E2 -25236.282} C_VEL
LIN {X 0,Y 173.22,Z 649.994,A -85,B 0,C 180,E1 -25238.644,E2 -25238.644} C_VEL
LIN {X 0,Y 163.61,Z 659.392,A -85,B 0,C 180,E1 -25242.183,E2 -25242.183} C_VEL
LIN {X 0,Y 155.826,Z 666.2,A -85,B 0,C 180,E1 -25245.646,E2 -25245.646} C_VEL
LIN {X 0,Y 147.904,Z 672.666,A -85,B 0,C 180,E1 -25250.096,E2 -25250.096} C_VEL
LIN {X 0,Y 141.012,Z 677.874,A -85,B 0,C 180,E1 -25255.028,E2 -25255.028} C_VEL
LIN {X 0,Y 136.602,Z 681.012,A -85,B 0,C 180,E1 -25259.099,E2 -25259.099} C_VEL
LIN {X 0,Y 133.96,Z 682.44,A -85,B 0,C 180,E1 -25261.267,E2 -25261.267} C_VEL
LIN {X 0,Y 128.368,Z 684.319,A -85,B 0,C 180,E1 -25264.754,E2 -25264.754} C_VEL
LIN {X 0,Y 124.121,Z 685.411,A -85,B 0,C 180,E1 -25267.76,E2 -25267.76} C_VEL
LIN {X 0,Y 121.88,Z 686.017,A -85,B 0,C 180,E1 -25270.295,E2 -25270.295} C_VEL
LIN {X 0,Y 121.435,Z 686.166,A -85,B 0,C 180,E1 -25271.195,E2 -25271.195} C_VEL
LIN {X 0,Y 120,Z 686.82,A -85,B 0,C 180,E1 -25276.45,E2 -25276.45} C_VEL
LIN {X 0,Y 119.513,Z 686.588,A -85,B 0,C 180,E1 -25283.244,E2 -25283.244} C_VEL
LIN {X 0,Y 119.728,Z 686.061,A -85,B 0,C 180,E1 -25286.633,E2 -25286.633} C_VEL
LIN {X 0,Y 119.998,Z 685.232,A -85,B 0,C 180,E1 -25289.999,E2 -25289.999} C_VEL
LIN {X 0,Y 119.753,Z 683.796,A -85,B 0,C 180,E1 -25293.912,E2 -25293.912} C_VEL
LIN {X 0,Y 119.752,Z 680.588,A -85,B 0,C 180,E1 -25300.139,E2 -25300.139} C_VEL
LIN {X 0,Y 120.901,Z 675.734,A -85,B 0,C 180,E1 -25306.895,E2 -25306.895} C_VEL
LIN {X 0,Y 123.498,Z 669.35,A -85,B 0,C 180,E1 -25313.474,E2 -25313.474} C_VEL
LIN {X 0,Y 127.442,Z 661.239,A -85,B 0,C 180,E1 -25319.755,E2 -25319.755} C_VEL
LIN {X 0,Y 132.044,Z 652.549,A -85,B 0,C 180,E1 -25324.9,E2 -25324.9} C_VEL
LIN {X 0,Y 137.041,Z 642.914,A -85,B 0,C 180,E1 -25329.349,E2 -25329.349} C_VEL
LIN {X 0,Y 142.043,Z 633.197,A -85,B 0,C 180,E1 -25332.867,E2 -25332.867} C_VEL
LIN {X 0,Y 148.037,Z 620.676,A -85,B 0,C 180,E1 -25336.383,E2 -25336.383} C_VEL
LIN {X 0,Y 153.459,Z 608.167,A -85,B 0,C 180,E1 -25339.081,E2 -25339.081} C_VEL
LIN {X 0,Y 158.577,Z 594.517,A -85,B 0,C 180,E1 -25341.362,E2 -25341.362} C_VEL
LIN {X 0,Y 163.171,Z 580.104,A -85,B 0,C 180,E1 -25343.184,E2 -25343.184} C_VEL
LIN {X 0,Y 167.115,Z 565.106,A -85,B 0,C 180,E1 -25344.567,E2 -25344.567} C_VEL
LIN {X 0,Y 170.106,Z 549.783,A -85,B 0,C 180,E1 -25345.588,E2 -25345.588} C_VEL
LIN {X 0,Y 172.247,Z 532.519,A -85,B 0,C 180,E1 -25346.366,E2 -25346.366} C_VEL
LIN {X 0,Y 177.775,Z 476.183,A -85,B 0,C 180,E1 -25348.42,E2 -25348.42} C_VEL
LIN {X 0,Y 172.567,Z 462.139,A -85,B 0,C 180,E1 -25351.328,E2 -25351.328} C_VEL
LIN {X 0,Y 166.79,Z 448.306,A -85,B 0,C 180,E1 -25354.768,E2 -25354.768} C_VEL
LIN {X 0,Y 161.724,Z 437.345,A -85,B 0,C 180,E1 -25358.101,E2 -25358.101} C_VEL
LIN {X 0,Y 159.084,Z 432.534,A -85,B 0,C 180,E1 -25359.893,E2 -25359.893} C_VEL
LIN {X 0,Y 153.843,Z 424.526,A -85,B 0,C 180,E1 -25363.77,E2 -25363.77} C_VEL
LIN {X 0,Y 150.742,Z 420.01,A -85,B 0,C 180,E1 -25366.3,E2 -25366.3} C_VEL
LIN {X 0,Y 148.551,Z 416.848,A -85,B 0,C 180,E1 -25368.274,E2 -25368.274} C_VEL
LIN {X 0,Y 145.405,Z 412.23,A -85,B 0,C 180,E1 -25371.457,E2 -25371.457} C_VEL
LIN {X 0,Y 142.678,Z 408.547,A -85,B 0,C 180,E1 -25374.525,E2 -25374.525} C_VEL
LIN {X 0,Y 141.8,Z 407.516,A -85,B 0,C 180,E1 -25375.604,E2 -25375.604} C_VEL
LIN {X 0,Y 139.656,Z 405.104,A -85,B 0,C 180,E1 -25378.49,E2 -25378.49} C_VEL
LIN {X 0,Y 138.335,Z 402.361,A -85,B 0,C 180,E1 -25380.729,E2 -25380.729} C_VEL
LIN {X 0,Y 135.44,Z 400.333,A -85,B 0,C 180,E1 -25385.958,E2 -25385.958} C_VEL
LIN {X 0,Y 134.213,Z 397.96,A -85,B 0,C 180,E1 -25389.415,E2 -25389.415} C_VEL
LIN {X 0,Y 133.888,Z 397.031,A -85,B 0,C 180,E1 -25390.712,E2 -25390.712} C_VEL
LIN {X 0,Y 132.318,Z 396.681,A -85,B 0,C 180,E1 -25401.828,E2 -25401.828} C_VEL
LIN {X 0,Y 133.599,Z 397.191,A -85,B 0,C 180,E1 -25409.551,E2 -25409.551} C_VEL
LIN {X 0,Y 135.192,Z 400.762,A -85,B 0,C 180,E1 -25414.88,E2 -25414.88} C_VEL
LIN {X 0,Y 137.971,Z 403.065,A -85,B 0,C 180,E1 -25420.081,E2 -25420.081} C_VEL
LIN {X 0,Y 139.78,Z 406.122,A -85,B 0,C 180,E1 -25423.022,E2 -25423.022} C_VEL
LIN {X 0,Y 142.139,Z 408.452,A -85,B 0,C 180,E1 -25426.059,E2 -25426.059} C_VEL
LIN {X 0,Y 144.651,Z 412.046,A -85,B 0,C 180,E1 -25429.029,E2 -25429.029} C_VEL
LIN {X 0,Y 145.987,Z 413.509,A -85,B 0,C 180,E1 -25430.379,E2 -25430.379} C_VEL
LIN {X 0,Y 149.788,Z 418.785,A -85,B 0,C 180,E1 -25434.037,E2 -25434.037} C_VEL
LIN {X 0,Y 153.225,Z 423.77,A -85,B 0,C 180,E1 -25436.923,E2 -25436.923} C_VEL
LIN {X 0,Y 157.396,Z 429.926,A -85,B 0,C 180,E1 -25440.068,E2 -25440.068} C_VEL
LIN {X 0,Y 163.102,Z 438.994,A -85,B 0,C 180,E1 -25443.863,E2 -25443.863} C_VEL
LIN {X 0,Y 170.231,Z 451.202,A -85,B 0,C 180,E1 -25448.051,E2 -25448.051} C_VEL
LIN {X 0,Y 177.952,Z 466.518,A -85,B 0,C 180,E1 -25452.091,E2 -25452.091} C_VEL
LIN {X 0,Y 171.783,Z 528.774,A -85,B 0,C 180,E1 -25454.427,E2 -25454.427} C_VEL
LIN {X 0,Y 169.308,Z 544.18,A -85,B 0,C 180,E1 -25455.349,E2 -25455.349} C_VEL
LIN {X 0,Y 166.109,Z 559.321,A -85,B 0,C 180,E1 -25456.69,E2 -25456.69} C_VEL
LIN {X 0,Y 161.963,Z 574.198,A -85,B 0,C 180,E1 -25458.424,E2 -25458.424} C_VEL
LIN {X 0,Y 157.312,Z 588.206,A -85,B 0,C 180,E1 -25460.587,E2 -25460.587} C_VEL
LIN {X 0,Y 152.411,Z 600.776,A -85,B 0,C 180,E1 -25463.049,E2 -25463.049} C_VEL
LIN {X 0,Y 146.752,Z 613.553,A -85,B 0,C 180,E1 -25466.261,E2 -25466.261} C_VEL
LIN {X 0,Y 141.191,Z 625.066,A -85,B 0,C 180,E1 -25470.001,E2 -25470.001} C_VEL
LIN {X 0,Y 135.642,Z 635.733,A -85,B 0,C 180,E1 -25474.459,E2 -25474.459} C_VEL
LIN {X 0,Y 130.832,Z 644.697,A -85,B 0,C 180,E1 -25479.275,E2 -25479.275} C_VEL
LIN {X 0,Y 126.809,Z 652.255,A -85,B 0,C 180,E1 -25484.443,E2 -25484.443} C_VEL
LIN {X 0,Y 123.661,Z 658.523,A -85,B 0,C 180,E1 -25489.939,E2 -25489.939} C_VEL
LIN {X 0,Y 121.373,Z 663.678,A -85,B 0,C 180,E1 -25495.741,E2 -25495.741} C_VEL
LIN {X 0,Y 119.802,Z 667.862,A -85,B 0,C 180,E1 -25501.87,E2 -25501.87} C_VEL
LIN {X 0,Y 119.238,Z 670.085,A -85,B 0,C 180,E1 -25506.117,E2 -25506.117} C_VEL
LIN {X 0,Y 119.148,Z 671.865,A -85,B 0,C 180,E1 -25510.456,E2 -25510.456} C_VEL
LIN {X 0,Y 119.589,Z 673.279,A -85,B 0,C 180,E1 -25515.151,E2 -25515.151} C_VEL
LIN {X 0,Y 120.582,Z 674.167,A -85,B 0,C 180,E1 -25520.123,E2 -25520.123} C_VEL
LIN {X 0,Y 122.2,Z 674.438,A -85,B 0,C 180,E1 -25524.89,E2 -25524.89} C_VEL
LIN {X 0,Y 124.477,Z 674.172,A -85,B 0,C 180,E1 -25529.458,E2 -25529.458} C_VEL
LIN {X 0,Y 127.317,Z 673.398,A -85,B 0,C 180,E1 -25533.792,E2 -25533.792} C_VEL
LIN {X 0,Y 130.742,Z 672.067,A -85,B 0,C 180,E1 -25537.895,E2 -25537.895} C_VEL
LIN {X 0,Y 134.717,Z 670.196,A -85,B 0,C 180,E1 -25541.758,E2 -25541.758} C_VEL
LIN {X 0,Y 141.514,Z 666.515,A -85,B 0,C 180,E1 -25547.006,E2 -25547.006} C_VEL
LIN {X 0,Y 149.665,Z 661.381,A -85,B 0,C 180,E1 -25551.901,E2 -25551.901} C_VEL
LIN {X 0,Y 158.669,Z 654.855,A -85,B 0,C 180,E1 -25556.191,E2 -25556.191} C_VEL
LIN {X 0,Y 168.675,Z 646.501,A -85,B 0,C 180,E1 -25560.121,E2 -25560.121} C_VEL
LIN {X 0,Y 177.481,Z 638.156,A -85,B 0,C 180,E1 -25563.001,E2 -25563.001} C_VEL
LIN {X 0,Y 186.527,Z 628.347,A -85,B 0,C 180,E1 -25565.549,E2 -25565.549} C_VEL
LIN {X 0,Y 195.865,Z 616.735,A -85,B 0,C 180,E1 -25567.82,E2 -25567.82} C_VEL
LIN {X 0,Y 203.693,Z 605.404,A -85,B 0,C 180,E1 -25569.533,E2 -25569.533} C_VEL
LIN {X 0,Y 210.789,Z 593.338,A -85,B 0,C 180,E1 -25570.994,E2 -25570.994} C_VEL
LIN {X 0,Y 217.811,Z 579.175,A -85,B 0,C 180,E1 -25572.298,E2 -25572.298} C_VEL
LIN {X 0,Y 223.757,Z 564.314,A -85,B 0,C 180,E1 -25573.366,E2 -25573.366} C_VEL
LIN {X 0,Y 228.484,Z 548.936,A -85,B 0,C 180,E1 -25574.178,E2 -25574.178} C_VEL
LIN {X 0,Y 231.881,Z 533.614,A -85,B 0,C 180,E1 -25574.729,E2 -25574.729} C_VEL
LIN {X 0,Y 236.118,Z 504.595,A -85,B 0,C 180,E1 -25575.538,E2 -25575.538} C_VEL
LIN {X 0,Y 235.622,Z 502.51,A -85,B 0,C 180,E1 -25579.153,E2 -25579.153} C_VEL
LIN {X 0,Y 235.591,Z 503.401,A -85,B 0,C 180,E1 -25580.88,E2 -25580.88} C_VEL
LIN {X 0,Y 235.804,Z 506.43,A -85,B 0,C 180,E1 -25583.493,E2 -25583.493} C_VEL
LIN {X 0,Y 235.87,Z 507.082,A -85,B 0,C 180,E1 -25583.871,E2 -25583.871} C_VEL
LIN {X 0,Y 231.167,Z 538.494,A -85,B 0,C 180,E1 -25584.66,E2 -25584.66} C_VEL
LIN {X 0,Y 227.855,Z 552.901,A -85,B 0,C 180,E1 -25585.107,E2 -25585.107} C_VEL
LIN {X 0,Y 223.231,Z 567.63,A -85,B 0,C 180,E1 -25585.682,E2 -25585.682} C_VEL
LIN {X 0,Y 216.982,Z 583.09,A -85,B 0,C 180,E1 -25586.52,E2 -25586.52} C_VEL
LIN {X 0,Y 210.088,Z 597.071,A -85,B 0,C 180,E1 -25587.563,E2 -25587.563} C_VEL
LIN {X 0,Y 202.5,Z 609.951,A -85,B 0,C 180,E1 -25588.795,E2 -25588.795} C_VEL
LIN {X 0,Y 193.557,Z 622.95,A -85,B 0,C 180,E1 -25590.517,E2 -25590.517} C_VEL
LIN {X 0,Y 184.595,Z 634.232,A -85,B 0,C 180,E1 -25592.499,E2 -25592.499} C_VEL
LIN {X 0,Y 175.538,Z 644.314,A -85,B 0,C 180,E1 -25594.838,E2 -25594.838} C_VEL
LIN {X 0,Y 168.918,Z 650.934,A -85,B 0,C 180,E1 -25596.781,E2 -25596.781} C_VEL
LIN {X 0,Y 158.955,Z 660.007,A -85,B 0,C 180,E1 -25600.297,E2 -25600.297} C_VEL
LIN {X 0,Y 150.84,Z 666.691,A -85,B 0,C 180,E1 -25603.763,E2 -25603.763} C_VEL
LIN {X 0,Y 142.498,Z 672.951,A -85,B 0,C 180,E1 -25608.253,E2 -25608.253} C_VEL
LIN {X 0,Y 135.209,Z 677.952,A -85,B 0,C 180,E1 -25613.289,E2 -25613.289} C_VEL
LIN {X 0,Y 130.089,Z 681.253,A -85,B 0,C 180,E1 -25617.91,E2 -25617.91} C_VEL
LIN {X 0,Y 125.1,Z 684.224,A -85,B 0,C 180,E1 -25624.007,E2 -25624.007} C_VEL
LIN {X 0,Y 121.435,Z 686.166,A -85,B 0,C 180,E1 -25631.195,E2 -25631.195} C_VEL
LIN {X 0,Y 119.871,Z 686.563,A -85,B 0,C 180,E1 -25633.895,E2 -25633.895} C_VEL
LIN {X 0,Y 116.126,Z 686.607,A -85,B 0,C 180,E1 -25638.354,E2 -25638.354} C_VEL
LIN {X 0,Y 113.5,Z 686.211,A -85,B 0,C 180,E1 -25642.104,E2 -25642.104} C_VEL
LIN {X 0,Y 112.602,Z 685.714,A -85,B 0,C 180,E1 -25645.067,E2 -25645.067} C_VEL
LIN {X 0,Y 112.622,Z 685.531,A -85,B 0,C 180,E1 -25646.071,E2 -25646.071} C_VEL
LIN {X 0,Y 112.933,Z 684.575,A -85,B 0,C 180,E1 -25649.998,E2 -25649.998} C_VEL
LIN {X 0,Y 112.688,Z 683.229,A -85,B 0,C 180,E1 -25653.755,E2 -25653.755} C_VEL
LIN {X 0,Y 112.743,Z 679.724,A -85,B 0,C 180,E1 -25660.777,E2 -25660.777} C_VEL
LIN {X 0,Y 114.056,Z 674.72,A -85,B 0,C 180,E1 -25667.943,E2 -25667.943} C_VEL
LIN {X 0,Y 116.953,Z 668.184,A -85,B 0,C 180,E1 -25674.874,E2 -25674.874} C_VEL
LIN {X 0,Y 120.632,Z 661.052,A -85,B 0,C 180,E1 -25680.647,E2 -25680.647} C_VEL
